REGION Network 77: WR 40001 - SETUP WRITING
   RUNG wire#powerrail
      { S7_Templates := "SrcType := Int" } EQ_Contact(in1 := "IEC_Counter_0_DB".CV, in2 := 71)
      Move(in := 16#8101, out1 => "Modbus_Send_Receive"."40001")
      { S7_Templates := "[card := 0, word_type := UInt, dword_type := UDInt, byte_type := USInt, any_type := Variant]" } "Modbus_Master_DB".Modbus_Master(REQ := wire#w1, MB_ADDR := 1, MODE := 1, DATA_ADDR := 40001, DATA_LEN := 1, DATA_PTR := "Modbus_Send_Receive"."40001", DONE => "Modbus".Done, BUSY => "Modbus".Busy, ERROR => "Modbus".Error, STATUS => "Modbus".Status)
   END_RUNG
   RUNG wire#powerrail
      Contact( "Comm_ok" )
      { S7_Templates := "SrcType := Int" } EQ_Contact(in1 := "IEC_Counter_0_DB".CV, in2 := 71)
      I_Contact( "Modbus_Master_DB".BUSY )
   END_RUNG wire#w1
   // the same network as SCL:
   IF "IEC_Counter_0_DB".CV = 71 THEN
       "Modbus_Send_Receive"."40001" := 16#8101;
       "Modbus_Master_DB"(REQ := "Comm_ok" AND ("IEC_Counter_0_DB".CV = 71) AND NOT "Modbus_Master_DB".BUSY,   // Modbus_Master
                          MB_ADDR := 1,
                          MODE := 1,
                          DATA_ADDR := 40001,
                          DATA_LEN := 1,
                          DATA_PTR := "Modbus_Send_Receive"."40001",
                          DONE => "Modbus".Done,
                          BUSY => "Modbus".Busy,
                          ERROR => "Modbus".Error,
                          STATUS => "Modbus".Status);
   END_IF;
END_REGION

REGION Network 78: WR 42001 - STS ON/OFF
   RUNG wire#powerrail
      { S7_Templates := "SrcType := Int" } EQ_Contact(in1 := "IEC_Counter_0_DB".CV, in2 := 72)
      { S7_Templates := "[card := 0, word_type := UInt, dword_type := UDInt, byte_type := USInt, any_type := Variant]" } "Modbus_Master_DB".Modbus_Master(REQ := wire#w2, MB_ADDR := 1, MODE := 1, DATA_ADDR := 42001, DATA_LEN := 1, DATA_PTR := "Modbus_Send_Receive"."42001", DONE => "Modbus".Done, BUSY => "Modbus".Busy, ERROR => "Modbus".Error, STATUS => "Modbus".Status)
   END_RUNG
   RUNG wire#powerrail
      Contact( "Liga_01" )
      Move(in := 16#0001, out1 => "Modbus_Send_Receive"."42001")
      wire#w1
      Contact( "Comm_ok" )
      { S7_Templates := "SrcType := Int" } EQ_Contact(in1 := "IEC_Counter_0_DB".CV, in2 := 72)
      I_Contact( "Modbus_Master_DB".BUSY )
   END_RUNG wire#w2
   RUNG wire#powerrail
      Contact( "Desliga_01" )
      Move(in := 16#0000, out1 => "Modbus_Send_Receive"."42001")
   END_RUNG wire#w1
   // the same network as SCL:
   IF "Liga_01" THEN "Modbus_Send_Receive"."42001" := 16#0001; END_IF;
   IF "Desliga_01" THEN "Modbus_Send_Receive"."42001" := 16#0000; END_IF;
   IF "IEC_Counter_0_DB".CV = 72 THEN
       "Modbus_Master_DB"(REQ := ("Liga_01" OR "Desliga_01") AND "Comm_ok" AND ("IEC_Counter_0_DB".CV = 72) AND NOT "Modbus_Master_DB".BUSY,   // Modbus_Master
                          MB_ADDR := 1,
                          MODE := 1,
                          DATA_ADDR := 42001,
                          DATA_LEN := 1,
                          DATA_PTR := "Modbus_Send_Receive"."42001",
                          DONE => "Modbus".Done,
                          BUSY => "Modbus".Busy,
                          ERROR => "Modbus".Error,
                          STATUS => "Modbus".Status);
   END_IF;
END_REGION

REGION Network 79: WR 42002 - OPER MODE
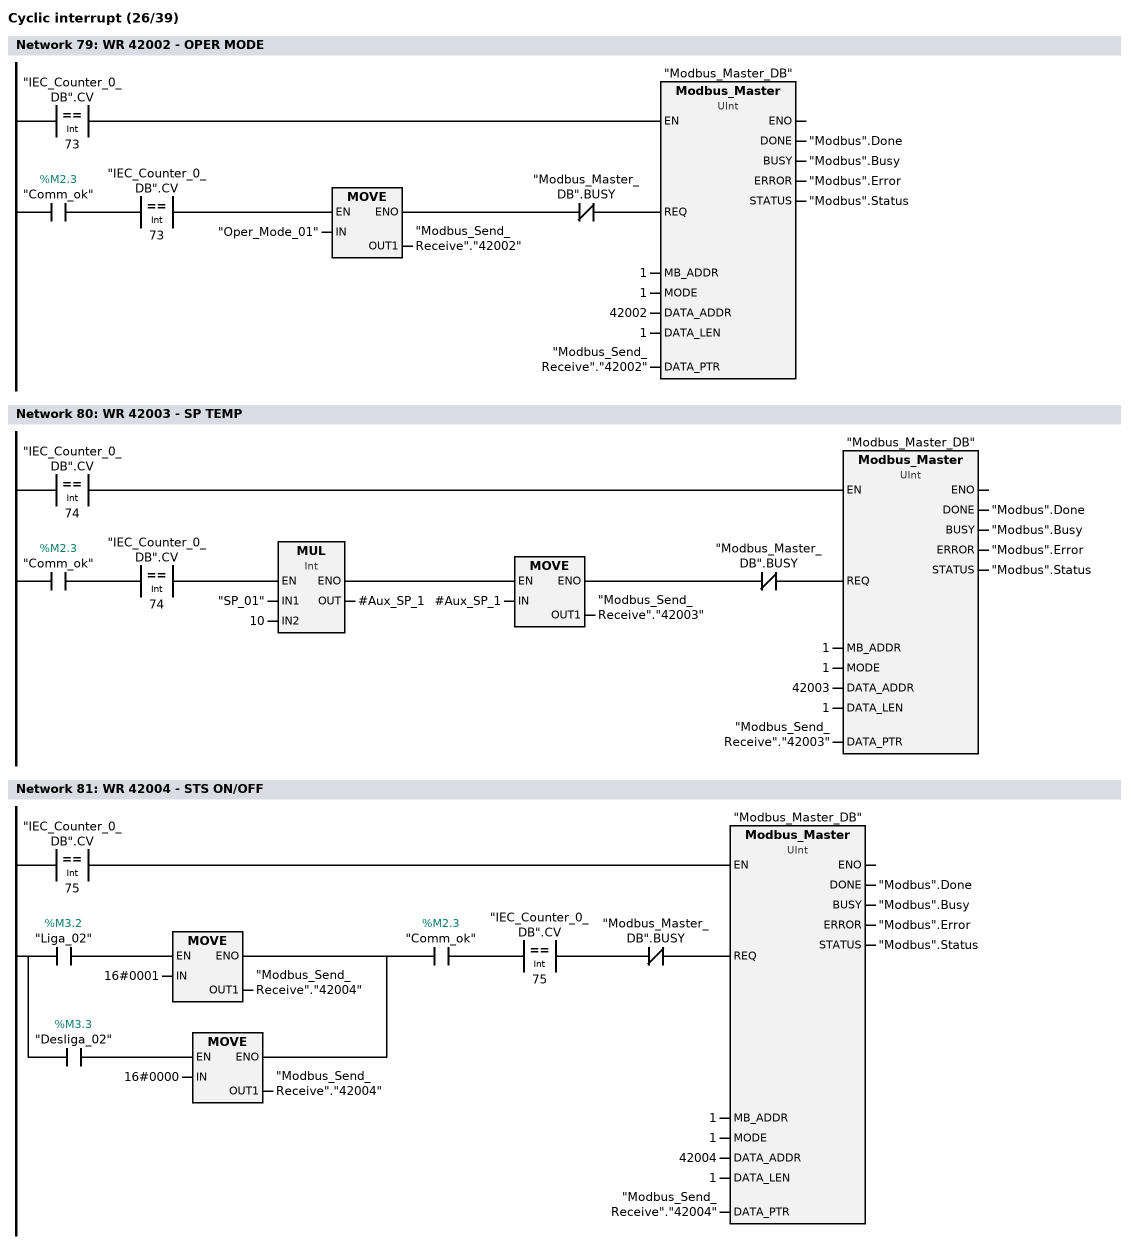
   RUNG wire#powerrail
      { S7_Templates := "SrcType := Int" } EQ_Contact(in1 := "IEC_Counter_0_DB".CV, in2 := 73)
      { S7_Templates := "[card := 0, word_type := UInt, dword_type := UDInt, byte_type := USInt, any_type := Variant]" } "Modbus_Master_DB".Modbus_Master(REQ := wire#w1, MB_ADDR := 1, MODE := 1, DATA_ADDR := 42002, DATA_LEN := 1, DATA_PTR := "Modbus_Send_Receive"."42002", DONE => "Modbus".Done, BUSY => "Modbus".Busy, ERROR => "Modbus".Error, STATUS => "Modbus".Status)
   END_RUNG
   RUNG wire#powerrail
      Contact( "Comm_ok" )
      { S7_Templates := "SrcType := Int" } EQ_Contact(in1 := "IEC_Counter_0_DB".CV, in2 := 73)
      Move(in := "Oper_Mode_01", out1 => "Modbus_Send_Receive"."42002")
      I_Contact( "Modbus_Master_DB".BUSY )
   END_RUNG wire#w1
   // the same network as SCL:
   #_w1 := "Comm_ok" AND ("IEC_Counter_0_DB".CV = 73);
   IF #_w1 THEN "Modbus_Send_Receive"."42002" := "Oper_Mode_01"; END_IF;
   IF "IEC_Counter_0_DB".CV = 73 THEN
       "Modbus_Master_DB"(REQ := #_w1 AND NOT "Modbus_Master_DB".BUSY,   // Modbus_Master
                          MB_ADDR := 1,
                          MODE := 1,
                          DATA_ADDR := 42002,
                          DATA_LEN := 1,
                          DATA_PTR := "Modbus_Send_Receive"."42002",
                          DONE => "Modbus".Done,
                          BUSY => "Modbus".Busy,
                          ERROR => "Modbus".Error,
                          STATUS => "Modbus".Status);
   END_IF;
END_REGION

REGION Network 80: WR 42003 - SP TEMP
   RUNG wire#powerrail
      { S7_Templates := "SrcType := Int" } EQ_Contact(in1 := "IEC_Counter_0_DB".CV, in2 := 74)
      { S7_Templates := "[card := 0, word_type := UInt, dword_type := UDInt, byte_type := USInt, any_type := Variant]" } "Modbus_Master_DB".Modbus_Master(REQ := wire#w1, MB_ADDR := 1, MODE := 1, DATA_ADDR := 42003, DATA_LEN := 1, DATA_PTR := "Modbus_Send_Receive"."42003", DONE => "Modbus".Done, BUSY => "Modbus".Busy, ERROR => "Modbus".Error, STATUS => "Modbus".Status)
   END_RUNG
   RUNG wire#powerrail
      Contact( "Comm_ok" )
      { S7_Templates := "SrcType := Int" } EQ_Contact(in1 := "IEC_Counter_0_DB".CV, in2 := 74)
      { S7_Templates := "SrcType := Int" } Mul(in1 := "SP_01", in2 := 10, out => #Aux_SP_1)
      Move(in := #Aux_SP_1, out1 => "Modbus_Send_Receive"."42003")
      I_Contact( "Modbus_Master_DB".BUSY )
   END_RUNG wire#w1
   // the same network as SCL:
   #_w1 := "Comm_ok" AND ("IEC_Counter_0_DB".CV = 74);
   IF #_w1 THEN
       #Aux_SP_1 := "SP_01" * 10;
       "Modbus_Send_Receive"."42003" := #Aux_SP_1;
   END_IF;
   IF "IEC_Counter_0_DB".CV = 74 THEN
       "Modbus_Master_DB"(REQ := #_w1 AND NOT "Modbus_Master_DB".BUSY,   // Modbus_Master
                          MB_ADDR := 1,
                          MODE := 1,
                          DATA_ADDR := 42003,
                          DATA_LEN := 1,
                          DATA_PTR := "Modbus_Send_Receive"."42003",
                          DONE => "Modbus".Done,
                          BUSY => "Modbus".Busy,
                          ERROR => "Modbus".Error,
                          STATUS => "Modbus".Status);
   END_IF;
END_REGION

REGION Network 81: WR 42004 - STS ON/OFF
   RUNG wire#powerrail
      { S7_Templates := "SrcType := Int" } EQ_Contact(in1 := "IEC_Counter_0_DB".CV, in2 := 75)
      { S7_Templates := "[card := 0, word_type := UInt, dword_type := UDInt, byte_type := USInt, any_type := Variant]" } "Modbus_Master_DB".Modbus_Master(REQ := wire#w2, MB_ADDR := 1, MODE := 1, DATA_ADDR := 42004, DATA_LEN := 1, DATA_PTR := "Modbus_Send_Receive"."42004", DONE => "Modbus".Done, BUSY => "Modbus".Busy, ERROR => "Modbus".Error, STATUS => "Modbus".Status)
   END_RUNG
   RUNG wire#powerrail
      Contact( "Liga_02" )
      Move(in := 16#0001, out1 => "Modbus_Send_Receive"."42004")
      wire#w1
      Contact( "Comm_ok" )
      { S7_Templates := "SrcType := Int" } EQ_Contact(in1 := "IEC_Counter_0_DB".CV, in2 := 75)
      I_Contact( "Modbus_Master_DB".BUSY )
   END_RUNG wire#w2
   RUNG wire#powerrail
      Contact( "Desliga_02" )
      Move(in := 16#0000, out1 => "Modbus_Send_Receive"."42004")
   END_RUNG wire#w1
   // the same network as SCL:
   IF "Liga_02" THEN "Modbus_Send_Receive"."42004" := 16#0001; END_IF;
   IF "Desliga_02" THEN "Modbus_Send_Receive"."42004" := 16#0000; END_IF;
   IF "IEC_Counter_0_DB".CV = 75 THEN
       "Modbus_Master_DB"(REQ := ("Liga_02" OR "Desliga_02") AND "Comm_ok" AND ("IEC_Counter_0_DB".CV = 75) AND NOT "Modbus_Master_DB".BUSY,   // Modbus_Master
                          MB_ADDR := 1,
                          MODE := 1,
                          DATA_ADDR := 42004,
                          DATA_LEN := 1,
                          DATA_PTR := "Modbus_Send_Receive"."42004",
                          DONE => "Modbus".Done,
                          BUSY => "Modbus".Busy,
                          ERROR => "Modbus".Error,
                          STATUS => "Modbus".Status);
   END_IF;
END_REGION

REGION Network 82: WR 42005 - OPER MODE
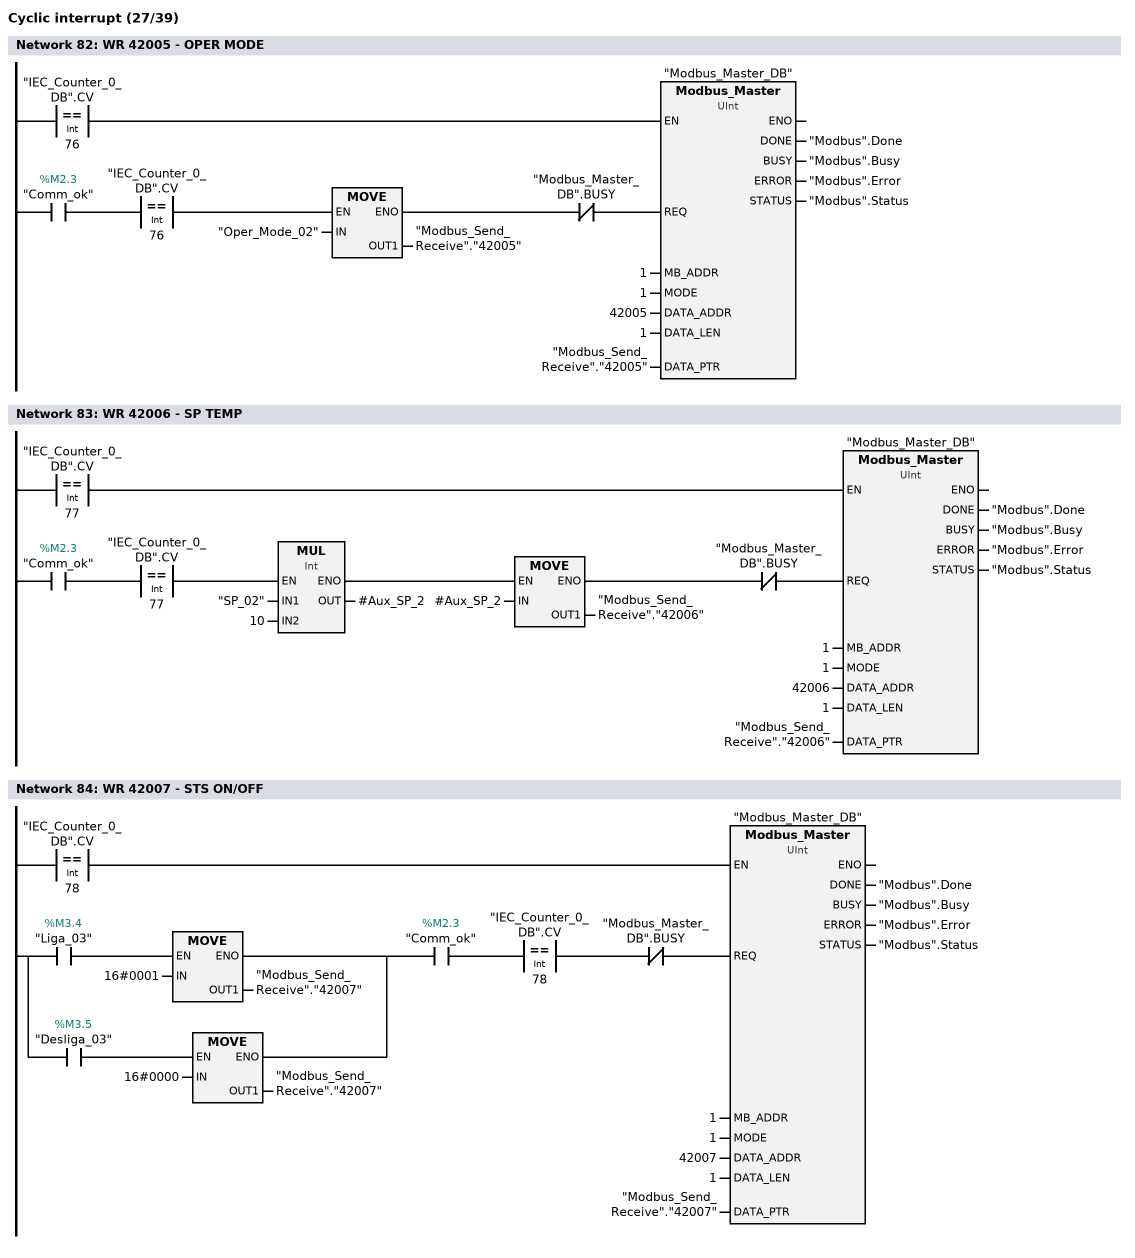
   RUNG wire#powerrail
      { S7_Templates := "SrcType := Int" } EQ_Contact(in1 := "IEC_Counter_0_DB".CV, in2 := 76)
      { S7_Templates := "[card := 0, word_type := UInt, dword_type := UDInt, byte_type := USInt, any_type := Variant]" } "Modbus_Master_DB".Modbus_Master(REQ := wire#w1, MB_ADDR := 1, MODE := 1, DATA_ADDR := 42005, DATA_LEN := 1, DATA_PTR := "Modbus_Send_Receive"."42005", DONE => "Modbus".Done, BUSY => "Modbus".Busy, ERROR => "Modbus".Error, STATUS => "Modbus".Status)
   END_RUNG
   RUNG wire#powerrail
      Contact( "Comm_ok" )
      { S7_Templates := "SrcType := Int" } EQ_Contact(in1 := "IEC_Counter_0_DB".CV, in2 := 76)
      Move(in := "Oper_Mode_02", out1 => "Modbus_Send_Receive"."42005")
      I_Contact( "Modbus_Master_DB".BUSY )
   END_RUNG wire#w1
   // the same network as SCL:
   #_w1 := "Comm_ok" AND ("IEC_Counter_0_DB".CV = 76);
   IF #_w1 THEN "Modbus_Send_Receive"."42005" := "Oper_Mode_02"; END_IF;
   IF "IEC_Counter_0_DB".CV = 76 THEN
       "Modbus_Master_DB"(REQ := #_w1 AND NOT "Modbus_Master_DB".BUSY,   // Modbus_Master
                          MB_ADDR := 1,
                          MODE := 1,
                          DATA_ADDR := 42005,
                          DATA_LEN := 1,
                          DATA_PTR := "Modbus_Send_Receive"."42005",
                          DONE => "Modbus".Done,
                          BUSY => "Modbus".Busy,
                          ERROR => "Modbus".Error,
                          STATUS => "Modbus".Status);
   END_IF;
END_REGION

REGION Network 83: WR 42006 - SP TEMP
   RUNG wire#powerrail
      { S7_Templates := "SrcType := Int" } EQ_Contact(in1 := "IEC_Counter_0_DB".CV, in2 := 77)
      { S7_Templates := "[card := 0, word_type := UInt, dword_type := UDInt, byte_type := USInt, any_type := Variant]" } "Modbus_Master_DB".Modbus_Master(REQ := wire#w1, MB_ADDR := 1, MODE := 1, DATA_ADDR := 42006, DATA_LEN := 1, DATA_PTR := "Modbus_Send_Receive"."42006", DONE => "Modbus".Done, BUSY => "Modbus".Busy, ERROR => "Modbus".Error, STATUS => "Modbus".Status)
   END_RUNG
   RUNG wire#powerrail
      Contact( "Comm_ok" )
      { S7_Templates := "SrcType := Int" } EQ_Contact(in1 := "IEC_Counter_0_DB".CV, in2 := 77)
      { S7_Templates := "SrcType := Int" } Mul(in1 := "SP_02", in2 := 10, out => #Aux_SP_2)
      Move(in := #Aux_SP_2, out1 => "Modbus_Send_Receive"."42006")
      I_Contact( "Modbus_Master_DB".BUSY )
   END_RUNG wire#w1
   // the same network as SCL:
   #_w1 := "Comm_ok" AND ("IEC_Counter_0_DB".CV = 77);
   IF #_w1 THEN
       #Aux_SP_2 := "SP_02" * 10;
       "Modbus_Send_Receive"."42006" := #Aux_SP_2;
   END_IF;
   IF "IEC_Counter_0_DB".CV = 77 THEN
       "Modbus_Master_DB"(REQ := #_w1 AND NOT "Modbus_Master_DB".BUSY,   // Modbus_Master
                          MB_ADDR := 1,
                          MODE := 1,
                          DATA_ADDR := 42006,
                          DATA_LEN := 1,
                          DATA_PTR := "Modbus_Send_Receive"."42006",
                          DONE => "Modbus".Done,
                          BUSY => "Modbus".Busy,
                          ERROR => "Modbus".Error,
                          STATUS => "Modbus".Status);
   END_IF;
END_REGION

REGION Network 84: WR 42007 - STS ON/OFF
   RUNG wire#powerrail
      { S7_Templates := "SrcType := Int" } EQ_Contact(in1 := "IEC_Counter_0_DB".CV, in2 := 78)
      { S7_Templates := "[card := 0, word_type := UInt, dword_type := UDInt, byte_type := USInt, any_type := Variant]" } "Modbus_Master_DB".Modbus_Master(REQ := wire#w2, MB_ADDR := 1, MODE := 1, DATA_ADDR := 42007, DATA_LEN := 1, DATA_PTR := "Modbus_Send_Receive"."42007", DONE => "Modbus".Done, BUSY => "Modbus".Busy, ERROR => "Modbus".Error, STATUS => "Modbus".Status)
   END_RUNG
   RUNG wire#powerrail
      Contact( "Liga_03" )
      Move(in := 16#0001, out1 => "Modbus_Send_Receive"."42007")
      wire#w1
      Contact( "Comm_ok" )
      { S7_Templates := "SrcType := Int" } EQ_Contact(in1 := "IEC_Counter_0_DB".CV, in2 := 78)
      I_Contact( "Modbus_Master_DB".BUSY )
   END_RUNG wire#w2
   RUNG wire#powerrail
      Contact( "Desliga_03" )
      Move(in := 16#0000, out1 => "Modbus_Send_Receive"."42007")
   END_RUNG wire#w1
   // the same network as SCL:
   IF "Liga_03" THEN "Modbus_Send_Receive"."42007" := 16#0001; END_IF;
   IF "Desliga_03" THEN "Modbus_Send_Receive"."42007" := 16#0000; END_IF;
   IF "IEC_Counter_0_DB".CV = 78 THEN
       "Modbus_Master_DB"(REQ := ("Liga_03" OR "Desliga_03") AND "Comm_ok" AND ("IEC_Counter_0_DB".CV = 78) AND NOT "Modbus_Master_DB".BUSY,   // Modbus_Master
                          MB_ADDR := 1,
                          MODE := 1,
                          DATA_ADDR := 42007,
                          DATA_LEN := 1,
                          DATA_PTR := "Modbus_Send_Receive"."42007",
                          DONE => "Modbus".Done,
                          BUSY => "Modbus".Busy,
                          ERROR => "Modbus".Error,
                          STATUS => "Modbus".Status);
   END_IF;
END_REGION

REGION Network 85: WR 42008 - OPER MODE
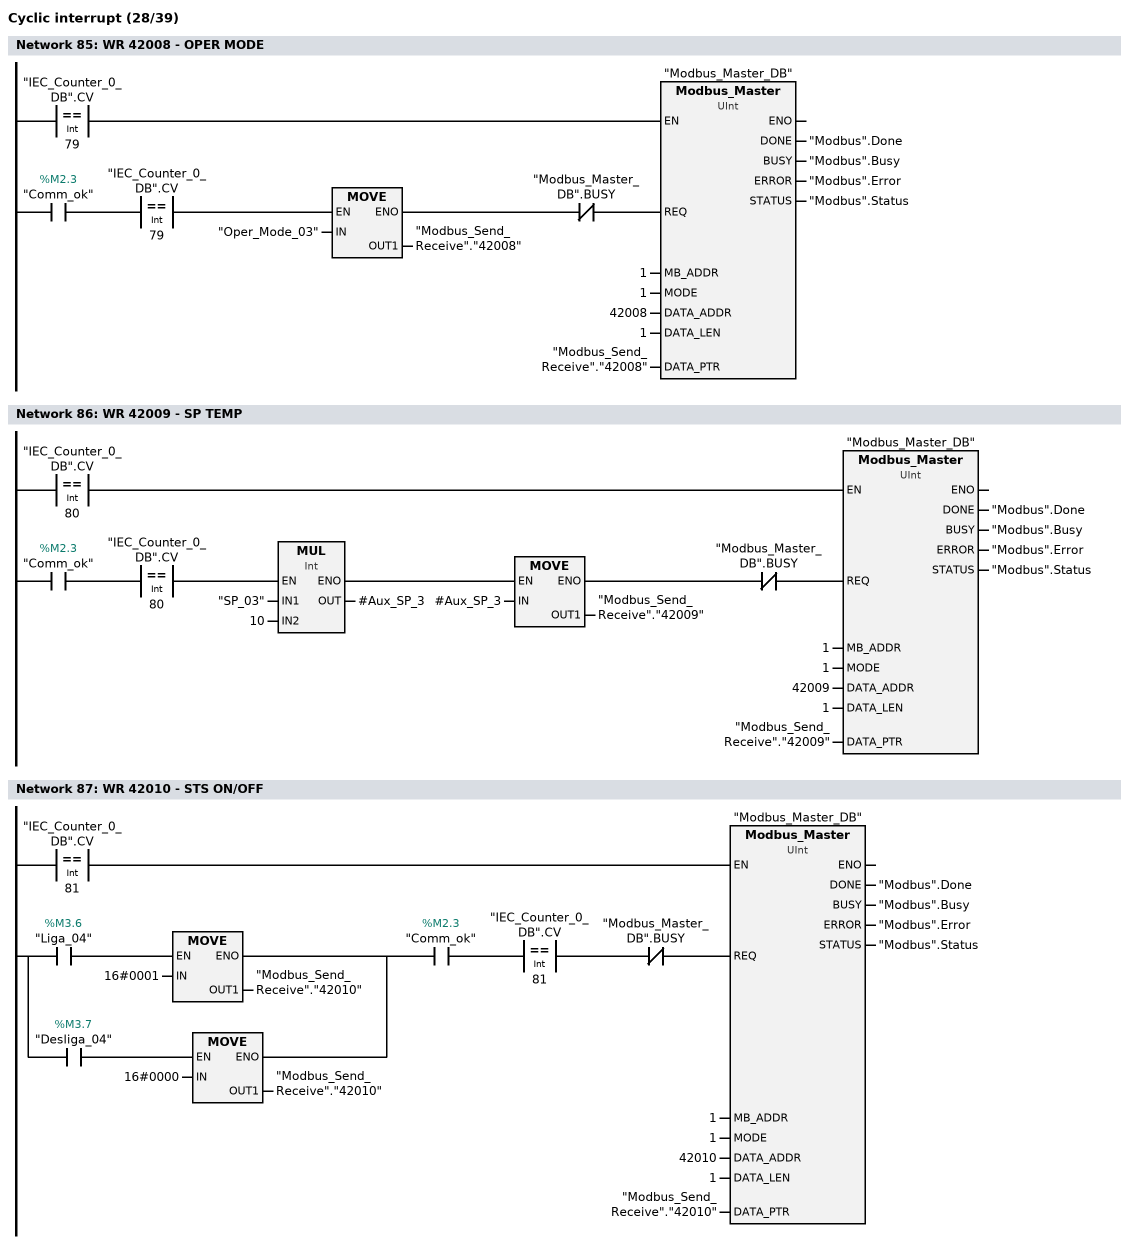
   RUNG wire#powerrail
      { S7_Templates := "SrcType := Int" } EQ_Contact(in1 := "IEC_Counter_0_DB".CV, in2 := 79)
      { S7_Templates := "[card := 0, word_type := UInt, dword_type := UDInt, byte_type := USInt, any_type := Variant]" } "Modbus_Master_DB".Modbus_Master(REQ := wire#w1, MB_ADDR := 1, MODE := 1, DATA_ADDR := 42008, DATA_LEN := 1, DATA_PTR := "Modbus_Send_Receive"."42008", DONE => "Modbus".Done, BUSY => "Modbus".Busy, ERROR => "Modbus".Error, STATUS => "Modbus".Status)
   END_RUNG
   RUNG wire#powerrail
      Contact( "Comm_ok" )
      { S7_Templates := "SrcType := Int" } EQ_Contact(in1 := "IEC_Counter_0_DB".CV, in2 := 79)
      Move(in := "Oper_Mode_03", out1 => "Modbus_Send_Receive"."42008")
      I_Contact( "Modbus_Master_DB".BUSY )
   END_RUNG wire#w1
   // the same network as SCL:
   #_w1 := "Comm_ok" AND ("IEC_Counter_0_DB".CV = 79);
   IF #_w1 THEN "Modbus_Send_Receive"."42008" := "Oper_Mode_03"; END_IF;
   IF "IEC_Counter_0_DB".CV = 79 THEN
       "Modbus_Master_DB"(REQ := #_w1 AND NOT "Modbus_Master_DB".BUSY,   // Modbus_Master
                          MB_ADDR := 1,
                          MODE := 1,
                          DATA_ADDR := 42008,
                          DATA_LEN := 1,
                          DATA_PTR := "Modbus_Send_Receive"."42008",
                          DONE => "Modbus".Done,
                          BUSY => "Modbus".Busy,
                          ERROR => "Modbus".Error,
                          STATUS => "Modbus".Status);
   END_IF;
END_REGION

REGION Network 86: WR 42009 - SP TEMP
   RUNG wire#powerrail
      { S7_Templates := "SrcType := Int" } EQ_Contact(in1 := "IEC_Counter_0_DB".CV, in2 := 80)
      { S7_Templates := "[card := 0, word_type := UInt, dword_type := UDInt, byte_type := USInt, any_type := Variant]" } "Modbus_Master_DB".Modbus_Master(REQ := wire#w1, MB_ADDR := 1, MODE := 1, DATA_ADDR := 42009, DATA_LEN := 1, DATA_PTR := "Modbus_Send_Receive"."42009", DONE => "Modbus".Done, BUSY => "Modbus".Busy, ERROR => "Modbus".Error, STATUS => "Modbus".Status)
   END_RUNG
   RUNG wire#powerrail
      Contact( "Comm_ok" )
      { S7_Templates := "SrcType := Int" } EQ_Contact(in1 := "IEC_Counter_0_DB".CV, in2 := 80)
      { S7_Templates := "SrcType := Int" } Mul(in1 := "SP_03", in2 := 10, out => #Aux_SP_3)
      Move(in := #Aux_SP_3, out1 => "Modbus_Send_Receive"."42009")
      I_Contact( "Modbus_Master_DB".BUSY )
   END_RUNG wire#w1
   // the same network as SCL:
   #_w1 := "Comm_ok" AND ("IEC_Counter_0_DB".CV = 80);
   IF #_w1 THEN
       #Aux_SP_3 := "SP_03" * 10;
       "Modbus_Send_Receive"."42009" := #Aux_SP_3;
   END_IF;
   IF "IEC_Counter_0_DB".CV = 80 THEN
       "Modbus_Master_DB"(REQ := #_w1 AND NOT "Modbus_Master_DB".BUSY,   // Modbus_Master
                          MB_ADDR := 1,
                          MODE := 1,
                          DATA_ADDR := 42009,
                          DATA_LEN := 1,
                          DATA_PTR := "Modbus_Send_Receive"."42009",
                          DONE => "Modbus".Done,
                          BUSY => "Modbus".Busy,
                          ERROR => "Modbus".Error,
                          STATUS => "Modbus".Status);
   END_IF;
END_REGION

REGION Network 87: WR 42010 - STS ON/OFF
   RUNG wire#powerrail
      { S7_Templates := "SrcType := Int" } EQ_Contact(in1 := "IEC_Counter_0_DB".CV, in2 := 81)
      { S7_Templates := "[card := 0, word_type := UInt, dword_type := UDInt, byte_type := USInt, any_type := Variant]" } "Modbus_Master_DB".Modbus_Master(REQ := wire#w2, MB_ADDR := 1, MODE := 1, DATA_ADDR := 42010, DATA_LEN := 1, DATA_PTR := "Modbus_Send_Receive"."42010", DONE => "Modbus".Done, BUSY => "Modbus".Busy, ERROR => "Modbus".Error, STATUS => "Modbus".Status)
   END_RUNG
   RUNG wire#powerrail
      Contact( "Liga_04" )
      Move(in := 16#0001, out1 => "Modbus_Send_Receive"."42010")
      wire#w1
      Contact( "Comm_ok" )
      { S7_Templates := "SrcType := Int" } EQ_Contact(in1 := "IEC_Counter_0_DB".CV, in2 := 81)
      I_Contact( "Modbus_Master_DB".BUSY )
   END_RUNG wire#w2
   RUNG wire#powerrail
      Contact( "Desliga_04" )
      Move(in := 16#0000, out1 => "Modbus_Send_Receive"."42010")
   END_RUNG wire#w1
   // the same network as SCL:
   IF "Liga_04" THEN "Modbus_Send_Receive"."42010" := 16#0001; END_IF;
   IF "Desliga_04" THEN "Modbus_Send_Receive"."42010" := 16#0000; END_IF;
   IF "IEC_Counter_0_DB".CV = 81 THEN
       "Modbus_Master_DB"(REQ := ("Liga_04" OR "Desliga_04") AND "Comm_ok" AND ("IEC_Counter_0_DB".CV = 81) AND NOT "Modbus_Master_DB".BUSY,   // Modbus_Master
                          MB_ADDR := 1,
                          MODE := 1,
                          DATA_ADDR := 42010,
                          DATA_LEN := 1,
                          DATA_PTR := "Modbus_Send_Receive"."42010",
                          DONE => "Modbus".Done,
                          BUSY => "Modbus".Busy,
                          ERROR => "Modbus".Error,
                          STATUS => "Modbus".Status);
   END_IF;
END_REGION

REGION Network 88: WR 42011 - OPER MODE
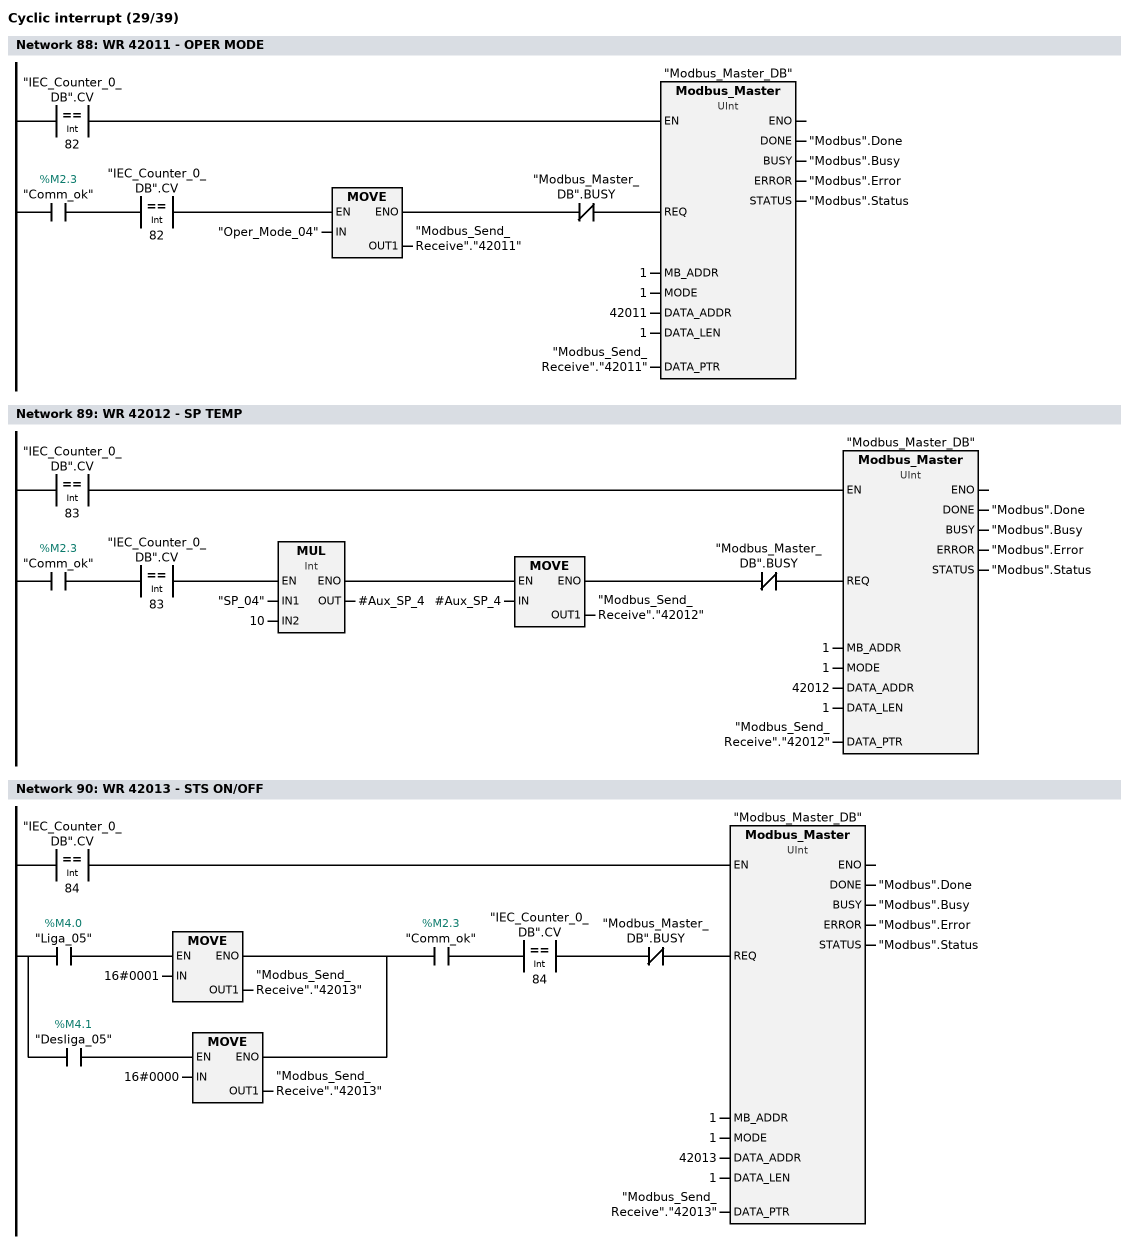
   RUNG wire#powerrail
      { S7_Templates := "SrcType := Int" } EQ_Contact(in1 := "IEC_Counter_0_DB".CV, in2 := 82)
      { S7_Templates := "[card := 0, word_type := UInt, dword_type := UDInt, byte_type := USInt, any_type := Variant]" } "Modbus_Master_DB".Modbus_Master(REQ := wire#w1, MB_ADDR := 1, MODE := 1, DATA_ADDR := 42011, DATA_LEN := 1, DATA_PTR := "Modbus_Send_Receive"."42011", DONE => "Modbus".Done, BUSY => "Modbus".Busy, ERROR => "Modbus".Error, STATUS => "Modbus".Status)
   END_RUNG
   RUNG wire#powerrail
      Contact( "Comm_ok" )
      { S7_Templates := "SrcType := Int" } EQ_Contact(in1 := "IEC_Counter_0_DB".CV, in2 := 82)
      Move(in := "Oper_Mode_04", out1 => "Modbus_Send_Receive"."42011")
      I_Contact( "Modbus_Master_DB".BUSY )
   END_RUNG wire#w1
   // the same network as SCL:
   #_w1 := "Comm_ok" AND ("IEC_Counter_0_DB".CV = 82);
   IF #_w1 THEN "Modbus_Send_Receive"."42011" := "Oper_Mode_04"; END_IF;
   IF "IEC_Counter_0_DB".CV = 82 THEN
       "Modbus_Master_DB"(REQ := #_w1 AND NOT "Modbus_Master_DB".BUSY,   // Modbus_Master
                          MB_ADDR := 1,
                          MODE := 1,
                          DATA_ADDR := 42011,
                          DATA_LEN := 1,
                          DATA_PTR := "Modbus_Send_Receive"."42011",
                          DONE => "Modbus".Done,
                          BUSY => "Modbus".Busy,
                          ERROR => "Modbus".Error,
                          STATUS => "Modbus".Status);
   END_IF;
END_REGION

REGION Network 89: WR 42012 - SP TEMP
   RUNG wire#powerrail
      { S7_Templates := "SrcType := Int" } EQ_Contact(in1 := "IEC_Counter_0_DB".CV, in2 := 83)
      { S7_Templates := "[card := 0, word_type := UInt, dword_type := UDInt, byte_type := USInt, any_type := Variant]" } "Modbus_Master_DB".Modbus_Master(REQ := wire#w1, MB_ADDR := 1, MODE := 1, DATA_ADDR := 42012, DATA_LEN := 1, DATA_PTR := "Modbus_Send_Receive"."42012", DONE => "Modbus".Done, BUSY => "Modbus".Busy, ERROR => "Modbus".Error, STATUS => "Modbus".Status)
   END_RUNG
   RUNG wire#powerrail
      Contact( "Comm_ok" )
      { S7_Templates := "SrcType := Int" } EQ_Contact(in1 := "IEC_Counter_0_DB".CV, in2 := 83)
      { S7_Templates := "SrcType := Int" } Mul(in1 := "SP_04", in2 := 10, out => #Aux_SP_4)
      Move(in := #Aux_SP_4, out1 => "Modbus_Send_Receive"."42012")
      I_Contact( "Modbus_Master_DB".BUSY )
   END_RUNG wire#w1
   // the same network as SCL:
   #_w1 := "Comm_ok" AND ("IEC_Counter_0_DB".CV = 83);
   IF #_w1 THEN
       #Aux_SP_4 := "SP_04" * 10;
       "Modbus_Send_Receive"."42012" := #Aux_SP_4;
   END_IF;
   IF "IEC_Counter_0_DB".CV = 83 THEN
       "Modbus_Master_DB"(REQ := #_w1 AND NOT "Modbus_Master_DB".BUSY,   // Modbus_Master
                          MB_ADDR := 1,
                          MODE := 1,
                          DATA_ADDR := 42012,
                          DATA_LEN := 1,
                          DATA_PTR := "Modbus_Send_Receive"."42012",
                          DONE => "Modbus".Done,
                          BUSY => "Modbus".Busy,
                          ERROR => "Modbus".Error,
                          STATUS => "Modbus".Status);
   END_IF;
END_REGION

REGION Network 90: WR 42013 - STS ON/OFF
   RUNG wire#powerrail
      { S7_Templates := "SrcType := Int" } EQ_Contact(in1 := "IEC_Counter_0_DB".CV, in2 := 84)
      { S7_Templates := "[card := 0, word_type := UInt, dword_type := UDInt, byte_type := USInt, any_type := Variant]" } "Modbus_Master_DB".Modbus_Master(REQ := wire#w2, MB_ADDR := 1, MODE := 1, DATA_ADDR := 42013, DATA_LEN := 1, DATA_PTR := "Modbus_Send_Receive"."42013", DONE => "Modbus".Done, BUSY => "Modbus".Busy, ERROR => "Modbus".Error, STATUS => "Modbus".Status)
   END_RUNG
   RUNG wire#powerrail
      Contact( "Liga_05" )
      Move(in := 16#0001, out1 => "Modbus_Send_Receive"."42013")
      wire#w1
      Contact( "Comm_ok" )
      { S7_Templates := "SrcType := Int" } EQ_Contact(in1 := "IEC_Counter_0_DB".CV, in2 := 84)
      I_Contact( "Modbus_Master_DB".BUSY )
   END_RUNG wire#w2
   RUNG wire#powerrail
      Contact( "Desliga_05" )
      Move(in := 16#0000, out1 => "Modbus_Send_Receive"."42013")
   END_RUNG wire#w1
   // the same network as SCL:
   IF "Liga_05" THEN "Modbus_Send_Receive"."42013" := 16#0001; END_IF;
   IF "Desliga_05" THEN "Modbus_Send_Receive"."42013" := 16#0000; END_IF;
   IF "IEC_Counter_0_DB".CV = 84 THEN
       "Modbus_Master_DB"(REQ := ("Liga_05" OR "Desliga_05") AND "Comm_ok" AND ("IEC_Counter_0_DB".CV = 84) AND NOT "Modbus_Master_DB".BUSY,   // Modbus_Master
                          MB_ADDR := 1,
                          MODE := 1,
                          DATA_ADDR := 42013,
                          DATA_LEN := 1,
                          DATA_PTR := "Modbus_Send_Receive"."42013",
                          DONE => "Modbus".Done,
                          BUSY => "Modbus".Busy,
                          ERROR => "Modbus".Error,
                          STATUS => "Modbus".Status);
   END_IF;
END_REGION

REGION Network 91: WR 42014 - OPER MODE
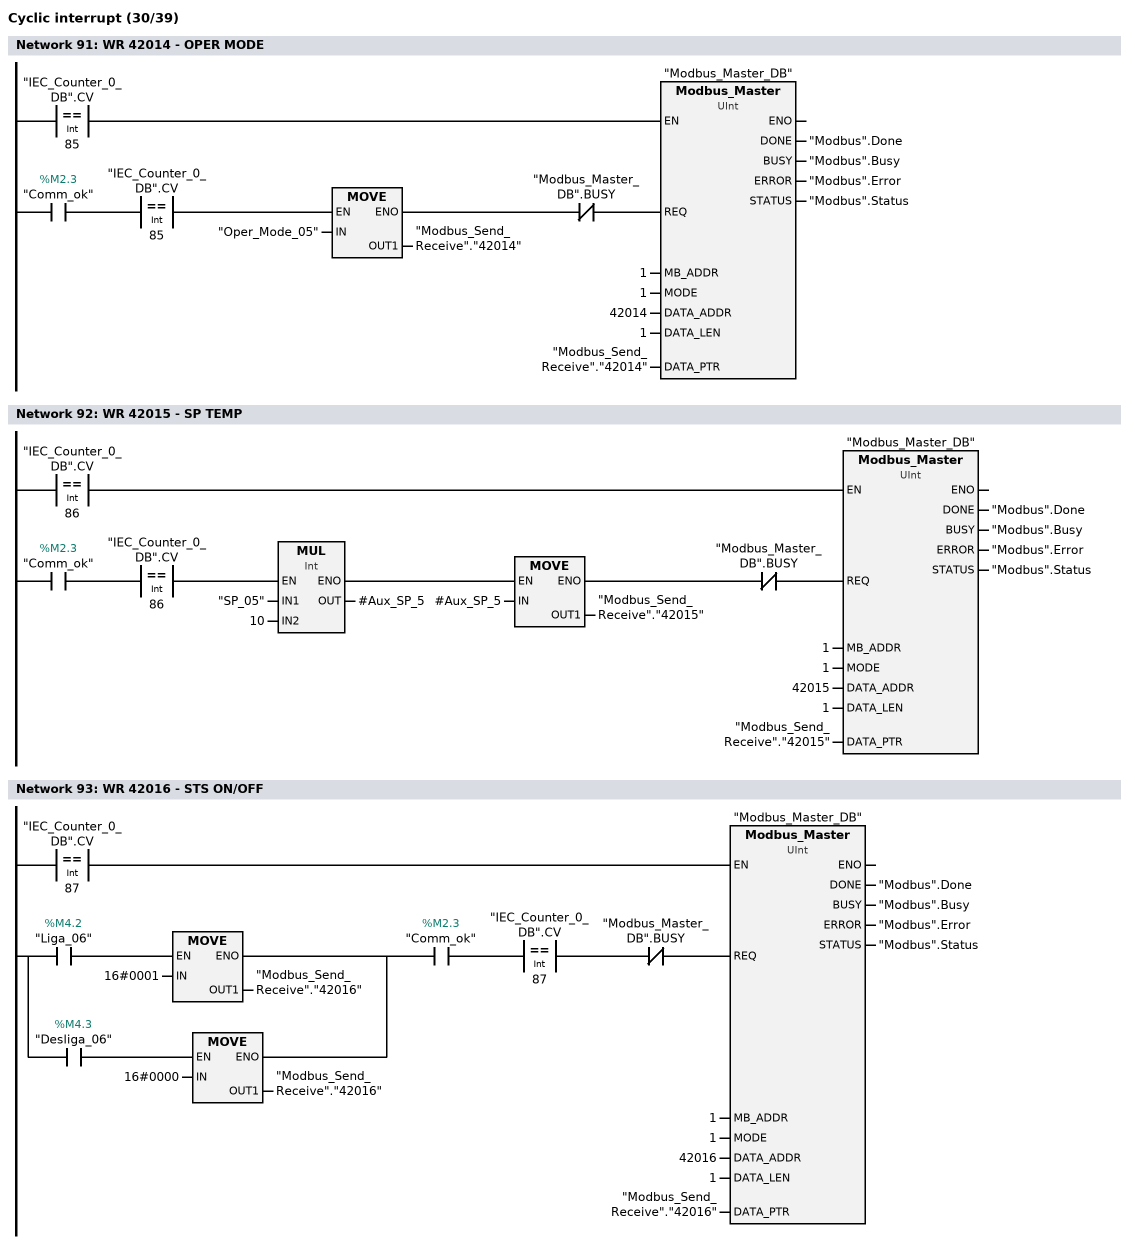
   RUNG wire#powerrail
      { S7_Templates := "SrcType := Int" } EQ_Contact(in1 := "IEC_Counter_0_DB".CV, in2 := 85)
      { S7_Templates := "[card := 0, word_type := UInt, dword_type := UDInt, byte_type := USInt, any_type := Variant]" } "Modbus_Master_DB".Modbus_Master(REQ := wire#w1, MB_ADDR := 1, MODE := 1, DATA_ADDR := 42014, DATA_LEN := 1, DATA_PTR := "Modbus_Send_Receive"."42014", DONE => "Modbus".Done, BUSY => "Modbus".Busy, ERROR => "Modbus".Error, STATUS => "Modbus".Status)
   END_RUNG
   RUNG wire#powerrail
      Contact( "Comm_ok" )
      { S7_Templates := "SrcType := Int" } EQ_Contact(in1 := "IEC_Counter_0_DB".CV, in2 := 85)
      Move(in := "Oper_Mode_05", out1 => "Modbus_Send_Receive"."42014")
      I_Contact( "Modbus_Master_DB".BUSY )
   END_RUNG wire#w1
   // the same network as SCL:
   #_w1 := "Comm_ok" AND ("IEC_Counter_0_DB".CV = 85);
   IF #_w1 THEN "Modbus_Send_Receive"."42014" := "Oper_Mode_05"; END_IF;
   IF "IEC_Counter_0_DB".CV = 85 THEN
       "Modbus_Master_DB"(REQ := #_w1 AND NOT "Modbus_Master_DB".BUSY,   // Modbus_Master
                          MB_ADDR := 1,
                          MODE := 1,
                          DATA_ADDR := 42014,
                          DATA_LEN := 1,
                          DATA_PTR := "Modbus_Send_Receive"."42014",
                          DONE => "Modbus".Done,
                          BUSY => "Modbus".Busy,
                          ERROR => "Modbus".Error,
                          STATUS => "Modbus".Status);
   END_IF;
END_REGION

REGION Network 92: WR 42015 - SP TEMP
   RUNG wire#powerrail
      { S7_Templates := "SrcType := Int" } EQ_Contact(in1 := "IEC_Counter_0_DB".CV, in2 := 86)
      { S7_Templates := "[card := 0, word_type := UInt, dword_type := UDInt, byte_type := USInt, any_type := Variant]" } "Modbus_Master_DB".Modbus_Master(REQ := wire#w1, MB_ADDR := 1, MODE := 1, DATA_ADDR := 42015, DATA_LEN := 1, DATA_PTR := "Modbus_Send_Receive"."42015", DONE => "Modbus".Done, BUSY => "Modbus".Busy, ERROR => "Modbus".Error, STATUS => "Modbus".Status)
   END_RUNG
   RUNG wire#powerrail
      Contact( "Comm_ok" )
      { S7_Templates := "SrcType := Int" } EQ_Contact(in1 := "IEC_Counter_0_DB".CV, in2 := 86)
      { S7_Templates := "SrcType := Int" } Mul(in1 := "SP_05", in2 := 10, out => #Aux_SP_5)
      Move(in := #Aux_SP_5, out1 => "Modbus_Send_Receive"."42015")
      I_Contact( "Modbus_Master_DB".BUSY )
   END_RUNG wire#w1
   // the same network as SCL:
   #_w1 := "Comm_ok" AND ("IEC_Counter_0_DB".CV = 86);
   IF #_w1 THEN
       #Aux_SP_5 := "SP_05" * 10;
       "Modbus_Send_Receive"."42015" := #Aux_SP_5;
   END_IF;
   IF "IEC_Counter_0_DB".CV = 86 THEN
       "Modbus_Master_DB"(REQ := #_w1 AND NOT "Modbus_Master_DB".BUSY,   // Modbus_Master
                          MB_ADDR := 1,
                          MODE := 1,
                          DATA_ADDR := 42015,
                          DATA_LEN := 1,
                          DATA_PTR := "Modbus_Send_Receive"."42015",
                          DONE => "Modbus".Done,
                          BUSY => "Modbus".Busy,
                          ERROR => "Modbus".Error,
                          STATUS => "Modbus".Status);
   END_IF;
END_REGION

REGION Network 93: WR 42016 - STS ON/OFF
   RUNG wire#powerrail
      { S7_Templates := "SrcType := Int" } EQ_Contact(in1 := "IEC_Counter_0_DB".CV, in2 := 87)
      { S7_Templates := "[card := 0, word_type := UInt, dword_type := UDInt, byte_type := USInt, any_type := Variant]" } "Modbus_Master_DB".Modbus_Master(REQ := wire#w2, MB_ADDR := 1, MODE := 1, DATA_ADDR := 42016, DATA_LEN := 1, DATA_PTR := "Modbus_Send_Receive"."42016", DONE => "Modbus".Done, BUSY => "Modbus".Busy, ERROR => "Modbus".Error, STATUS => "Modbus".Status)
   END_RUNG
   RUNG wire#powerrail
      Contact( "Liga_06" )
      Move(in := 16#0001, out1 => "Modbus_Send_Receive"."42016")
      wire#w1
      Contact( "Comm_ok" )
      { S7_Templates := "SrcType := Int" } EQ_Contact(in1 := "IEC_Counter_0_DB".CV, in2 := 87)
      I_Contact( "Modbus_Master_DB".BUSY )
   END_RUNG wire#w2
   RUNG wire#powerrail
      Contact( "Desliga_06" )
      Move(in := 16#0000, out1 => "Modbus_Send_Receive"."42016")
   END_RUNG wire#w1
   // the same network as SCL:
   IF "Liga_06" THEN "Modbus_Send_Receive"."42016" := 16#0001; END_IF;
   IF "Desliga_06" THEN "Modbus_Send_Receive"."42016" := 16#0000; END_IF;
   IF "IEC_Counter_0_DB".CV = 87 THEN
       "Modbus_Master_DB"(REQ := ("Liga_06" OR "Desliga_06") AND "Comm_ok" AND ("IEC_Counter_0_DB".CV = 87) AND NOT "Modbus_Master_DB".BUSY,   // Modbus_Master
                          MB_ADDR := 1,
                          MODE := 1,
                          DATA_ADDR := 42016,
                          DATA_LEN := 1,
                          DATA_PTR := "Modbus_Send_Receive"."42016",
                          DONE => "Modbus".Done,
                          BUSY => "Modbus".Busy,
                          ERROR => "Modbus".Error,
                          STATUS => "Modbus".Status);
   END_IF;
END_REGION

REGION Network 94: WR 42017 - OPER MODE
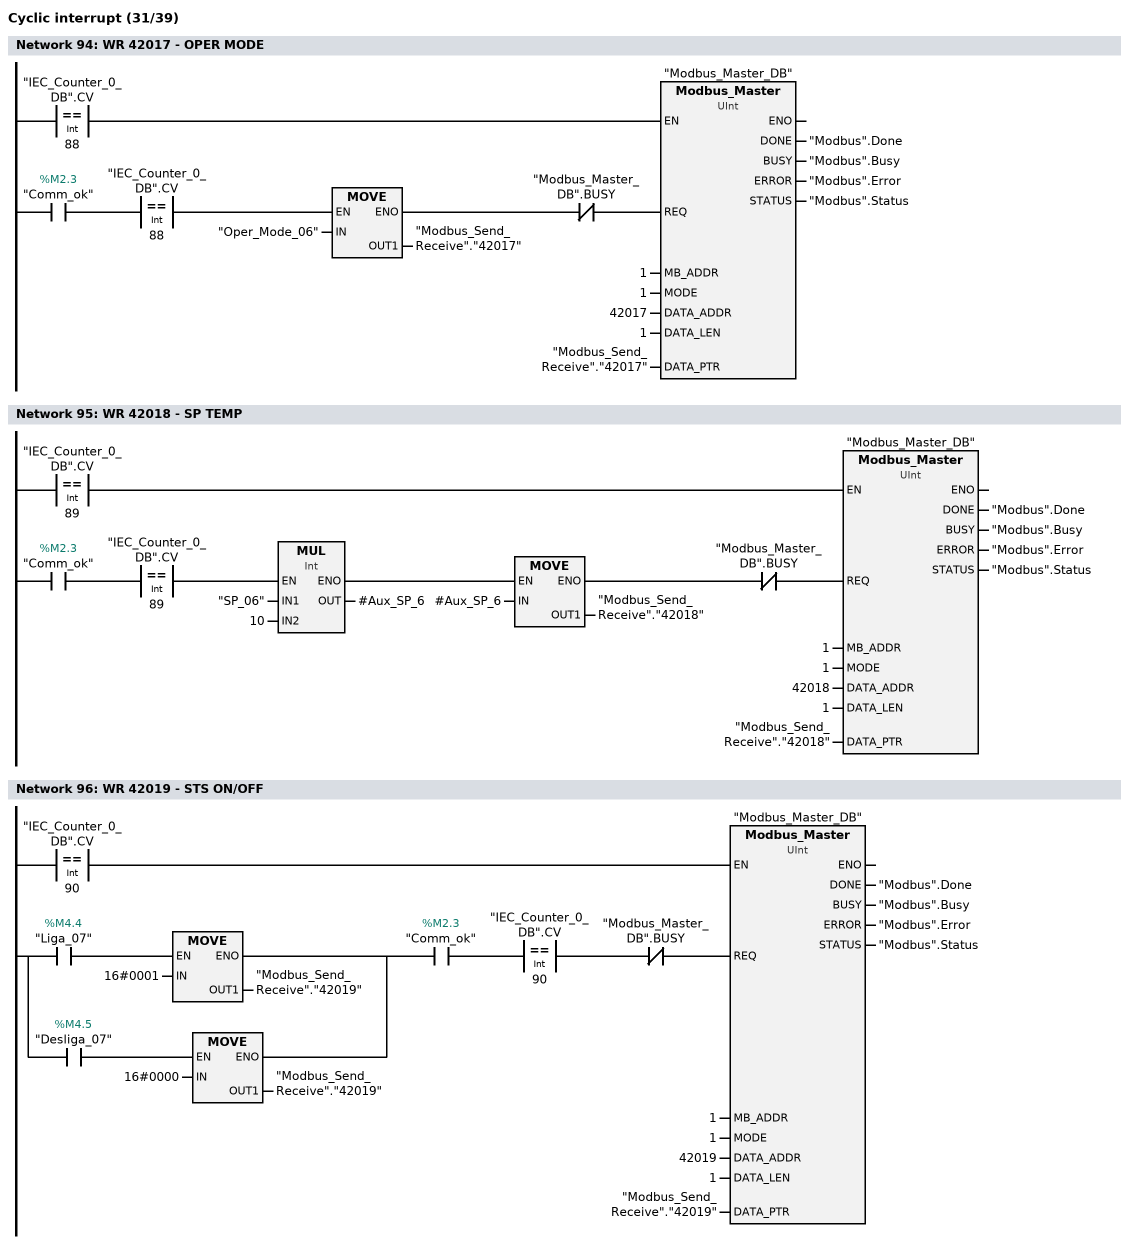
   RUNG wire#powerrail
      { S7_Templates := "SrcType := Int" } EQ_Contact(in1 := "IEC_Counter_0_DB".CV, in2 := 88)
      { S7_Templates := "[card := 0, word_type := UInt, dword_type := UDInt, byte_type := USInt, any_type := Variant]" } "Modbus_Master_DB".Modbus_Master(REQ := wire#w1, MB_ADDR := 1, MODE := 1, DATA_ADDR := 42017, DATA_LEN := 1, DATA_PTR := "Modbus_Send_Receive"."42017", DONE => "Modbus".Done, BUSY => "Modbus".Busy, ERROR => "Modbus".Error, STATUS => "Modbus".Status)
   END_RUNG
   RUNG wire#powerrail
      Contact( "Comm_ok" )
      { S7_Templates := "SrcType := Int" } EQ_Contact(in1 := "IEC_Counter_0_DB".CV, in2 := 88)
      Move(in := "Oper_Mode_06", out1 => "Modbus_Send_Receive"."42017")
      I_Contact( "Modbus_Master_DB".BUSY )
   END_RUNG wire#w1
   // the same network as SCL:
   #_w1 := "Comm_ok" AND ("IEC_Counter_0_DB".CV = 88);
   IF #_w1 THEN "Modbus_Send_Receive"."42017" := "Oper_Mode_06"; END_IF;
   IF "IEC_Counter_0_DB".CV = 88 THEN
       "Modbus_Master_DB"(REQ := #_w1 AND NOT "Modbus_Master_DB".BUSY,   // Modbus_Master
                          MB_ADDR := 1,
                          MODE := 1,
                          DATA_ADDR := 42017,
                          DATA_LEN := 1,
                          DATA_PTR := "Modbus_Send_Receive"."42017",
                          DONE => "Modbus".Done,
                          BUSY => "Modbus".Busy,
                          ERROR => "Modbus".Error,
                          STATUS => "Modbus".Status);
   END_IF;
END_REGION

REGION Network 95: WR 42018 - SP TEMP
   RUNG wire#powerrail
      { S7_Templates := "SrcType := Int" } EQ_Contact(in1 := "IEC_Counter_0_DB".CV, in2 := 89)
      { S7_Templates := "[card := 0, word_type := UInt, dword_type := UDInt, byte_type := USInt, any_type := Variant]" } "Modbus_Master_DB".Modbus_Master(REQ := wire#w1, MB_ADDR := 1, MODE := 1, DATA_ADDR := 42018, DATA_LEN := 1, DATA_PTR := "Modbus_Send_Receive"."42018", DONE => "Modbus".Done, BUSY => "Modbus".Busy, ERROR => "Modbus".Error, STATUS => "Modbus".Status)
   END_RUNG
   RUNG wire#powerrail
      Contact( "Comm_ok" )
      { S7_Templates := "SrcType := Int" } EQ_Contact(in1 := "IEC_Counter_0_DB".CV, in2 := 89)
      { S7_Templates := "SrcType := Int" } Mul(in1 := "SP_06", in2 := 10, out => #Aux_SP_6)
      Move(in := #Aux_SP_6, out1 => "Modbus_Send_Receive"."42018")
      I_Contact( "Modbus_Master_DB".BUSY )
   END_RUNG wire#w1
   // the same network as SCL:
   #_w1 := "Comm_ok" AND ("IEC_Counter_0_DB".CV = 89);
   IF #_w1 THEN
       #Aux_SP_6 := "SP_06" * 10;
       "Modbus_Send_Receive"."42018" := #Aux_SP_6;
   END_IF;
   IF "IEC_Counter_0_DB".CV = 89 THEN
       "Modbus_Master_DB"(REQ := #_w1 AND NOT "Modbus_Master_DB".BUSY,   // Modbus_Master
                          MB_ADDR := 1,
                          MODE := 1,
                          DATA_ADDR := 42018,
                          DATA_LEN := 1,
                          DATA_PTR := "Modbus_Send_Receive"."42018",
                          DONE => "Modbus".Done,
                          BUSY => "Modbus".Busy,
                          ERROR => "Modbus".Error,
                          STATUS => "Modbus".Status);
   END_IF;
END_REGION

REGION Network 96: WR 42019 - STS ON/OFF
   RUNG wire#powerrail
      { S7_Templates := "SrcType := Int" } EQ_Contact(in1 := "IEC_Counter_0_DB".CV, in2 := 90)
      { S7_Templates := "[card := 0, word_type := UInt, dword_type := UDInt, byte_type := USInt, any_type := Variant]" } "Modbus_Master_DB".Modbus_Master(REQ := wire#w2, MB_ADDR := 1, MODE := 1, DATA_ADDR := 42019, DATA_LEN := 1, DATA_PTR := "Modbus_Send_Receive"."42019", DONE => "Modbus".Done, BUSY => "Modbus".Busy, ERROR => "Modbus".Error, STATUS => "Modbus".Status)
   END_RUNG
   RUNG wire#powerrail
      Contact( "Liga_07" )
      Move(in := 16#0001, out1 => "Modbus_Send_Receive"."42019")
      wire#w1
      Contact( "Comm_ok" )
      { S7_Templates := "SrcType := Int" } EQ_Contact(in1 := "IEC_Counter_0_DB".CV, in2 := 90)
      I_Contact( "Modbus_Master_DB".BUSY )
   END_RUNG wire#w2
   RUNG wire#powerrail
      Contact( "Desliga_07" )
      Move(in := 16#0000, out1 => "Modbus_Send_Receive"."42019")
   END_RUNG wire#w1
   // the same network as SCL:
   IF "Liga_07" THEN "Modbus_Send_Receive"."42019" := 16#0001; END_IF;
   IF "Desliga_07" THEN "Modbus_Send_Receive"."42019" := 16#0000; END_IF;
   IF "IEC_Counter_0_DB".CV = 90 THEN
       "Modbus_Master_DB"(REQ := ("Liga_07" OR "Desliga_07") AND "Comm_ok" AND ("IEC_Counter_0_DB".CV = 90) AND NOT "Modbus_Master_DB".BUSY,   // Modbus_Master
                          MB_ADDR := 1,
                          MODE := 1,
                          DATA_ADDR := 42019,
                          DATA_LEN := 1,
                          DATA_PTR := "Modbus_Send_Receive"."42019",
                          DONE => "Modbus".Done,
                          BUSY => "Modbus".Busy,
                          ERROR => "Modbus".Error,
                          STATUS => "Modbus".Status);
   END_IF;
END_REGION

REGION Network 97: WR 42020 - OPER MODE
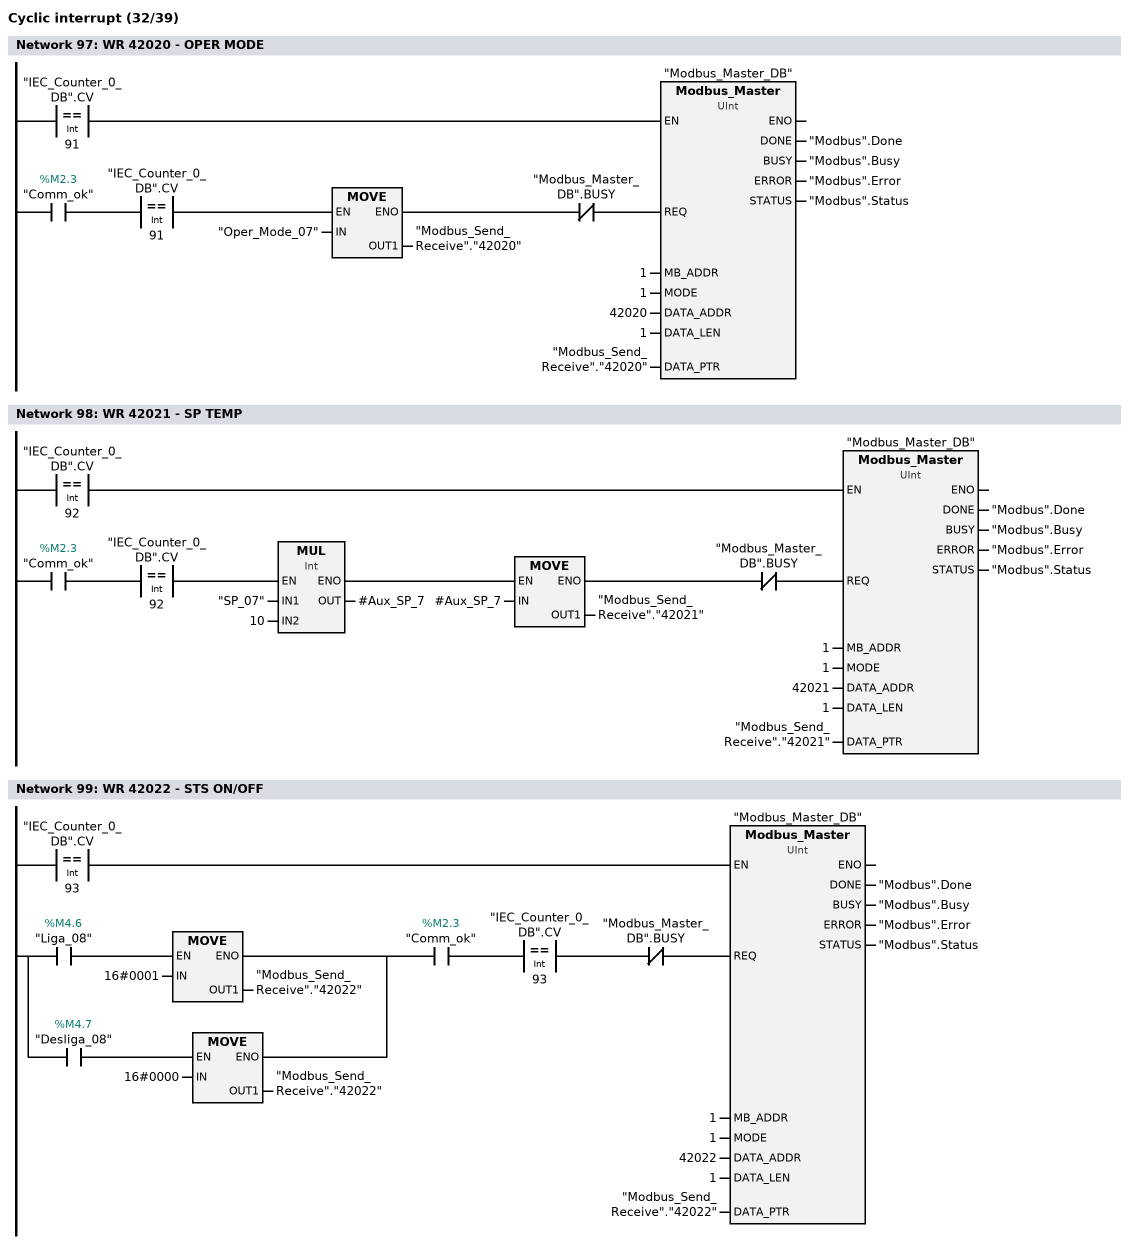
   RUNG wire#powerrail
      { S7_Templates := "SrcType := Int" } EQ_Contact(in1 := "IEC_Counter_0_DB".CV, in2 := 91)
      { S7_Templates := "[card := 0, word_type := UInt, dword_type := UDInt, byte_type := USInt, any_type := Variant]" } "Modbus_Master_DB".Modbus_Master(REQ := wire#w1, MB_ADDR := 1, MODE := 1, DATA_ADDR := 42020, DATA_LEN := 1, DATA_PTR := "Modbus_Send_Receive"."42020", DONE => "Modbus".Done, BUSY => "Modbus".Busy, ERROR => "Modbus".Error, STATUS => "Modbus".Status)
   END_RUNG
   RUNG wire#powerrail
      Contact( "Comm_ok" )
      { S7_Templates := "SrcType := Int" } EQ_Contact(in1 := "IEC_Counter_0_DB".CV, in2 := 91)
      Move(in := "Oper_Mode_07", out1 => "Modbus_Send_Receive"."42020")
      I_Contact( "Modbus_Master_DB".BUSY )
   END_RUNG wire#w1
   // the same network as SCL:
   #_w1 := "Comm_ok" AND ("IEC_Counter_0_DB".CV = 91);
   IF #_w1 THEN "Modbus_Send_Receive"."42020" := "Oper_Mode_07"; END_IF;
   IF "IEC_Counter_0_DB".CV = 91 THEN
       "Modbus_Master_DB"(REQ := #_w1 AND NOT "Modbus_Master_DB".BUSY,   // Modbus_Master
                          MB_ADDR := 1,
                          MODE := 1,
                          DATA_ADDR := 42020,
                          DATA_LEN := 1,
                          DATA_PTR := "Modbus_Send_Receive"."42020",
                          DONE => "Modbus".Done,
                          BUSY => "Modbus".Busy,
                          ERROR => "Modbus".Error,
                          STATUS => "Modbus".Status);
   END_IF;
END_REGION

REGION Network 98: WR 42021 - SP TEMP
   RUNG wire#powerrail
      { S7_Templates := "SrcType := Int" } EQ_Contact(in1 := "IEC_Counter_0_DB".CV, in2 := 92)
      { S7_Templates := "[card := 0, word_type := UInt, dword_type := UDInt, byte_type := USInt, any_type := Variant]" } "Modbus_Master_DB".Modbus_Master(REQ := wire#w1, MB_ADDR := 1, MODE := 1, DATA_ADDR := 42021, DATA_LEN := 1, DATA_PTR := "Modbus_Send_Receive"."42021", DONE => "Modbus".Done, BUSY => "Modbus".Busy, ERROR => "Modbus".Error, STATUS => "Modbus".Status)
   END_RUNG
   RUNG wire#powerrail
      Contact( "Comm_ok" )
      { S7_Templates := "SrcType := Int" } EQ_Contact(in1 := "IEC_Counter_0_DB".CV, in2 := 92)
      { S7_Templates := "SrcType := Int" } Mul(in1 := "SP_07", in2 := 10, out => #Aux_SP_7)
      Move(in := #Aux_SP_7, out1 => "Modbus_Send_Receive"."42021")
      I_Contact( "Modbus_Master_DB".BUSY )
   END_RUNG wire#w1
   // the same network as SCL:
   #_w1 := "Comm_ok" AND ("IEC_Counter_0_DB".CV = 92);
   IF #_w1 THEN
       #Aux_SP_7 := "SP_07" * 10;
       "Modbus_Send_Receive"."42021" := #Aux_SP_7;
   END_IF;
   IF "IEC_Counter_0_DB".CV = 92 THEN
       "Modbus_Master_DB"(REQ := #_w1 AND NOT "Modbus_Master_DB".BUSY,   // Modbus_Master
                          MB_ADDR := 1,
                          MODE := 1,
                          DATA_ADDR := 42021,
                          DATA_LEN := 1,
                          DATA_PTR := "Modbus_Send_Receive"."42021",
                          DONE => "Modbus".Done,
                          BUSY => "Modbus".Busy,
                          ERROR => "Modbus".Error,
                          STATUS => "Modbus".Status);
   END_IF;
END_REGION

REGION Network 99: WR 42022 - STS ON/OFF
   RUNG wire#powerrail
      { S7_Templates := "SrcType := Int" } EQ_Contact(in1 := "IEC_Counter_0_DB".CV, in2 := 93)
      { S7_Templates := "[card := 0, word_type := UInt, dword_type := UDInt, byte_type := USInt, any_type := Variant]" } "Modbus_Master_DB".Modbus_Master(REQ := wire#w2, MB_ADDR := 1, MODE := 1, DATA_ADDR := 42022, DATA_LEN := 1, DATA_PTR := "Modbus_Send_Receive"."42022", DONE => "Modbus".Done, BUSY => "Modbus".Busy, ERROR => "Modbus".Error, STATUS => "Modbus".Status)
   END_RUNG
   RUNG wire#powerrail
      Contact( "Liga_08" )
      Move(in := 16#0001, out1 => "Modbus_Send_Receive"."42022")
      wire#w1
      Contact( "Comm_ok" )
      { S7_Templates := "SrcType := Int" } EQ_Contact(in1 := "IEC_Counter_0_DB".CV, in2 := 93)
      I_Contact( "Modbus_Master_DB".BUSY )
   END_RUNG wire#w2
   RUNG wire#powerrail
      Contact( "Desliga_08" )
      Move(in := 16#0000, out1 => "Modbus_Send_Receive"."42022")
   END_RUNG wire#w1
   // the same network as SCL:
   IF "Liga_08" THEN "Modbus_Send_Receive"."42022" := 16#0001; END_IF;
   IF "Desliga_08" THEN "Modbus_Send_Receive"."42022" := 16#0000; END_IF;
   IF "IEC_Counter_0_DB".CV = 93 THEN
       "Modbus_Master_DB"(REQ := ("Liga_08" OR "Desliga_08") AND "Comm_ok" AND ("IEC_Counter_0_DB".CV = 93) AND NOT "Modbus_Master_DB".BUSY,   // Modbus_Master
                          MB_ADDR := 1,
                          MODE := 1,
                          DATA_ADDR := 42022,
                          DATA_LEN := 1,
                          DATA_PTR := "Modbus_Send_Receive"."42022",
                          DONE => "Modbus".Done,
                          BUSY => "Modbus".Busy,
                          ERROR => "Modbus".Error,
                          STATUS => "Modbus".Status);
   END_IF;
END_REGION

REGION Network 100: WR 42023 - OPER MODE
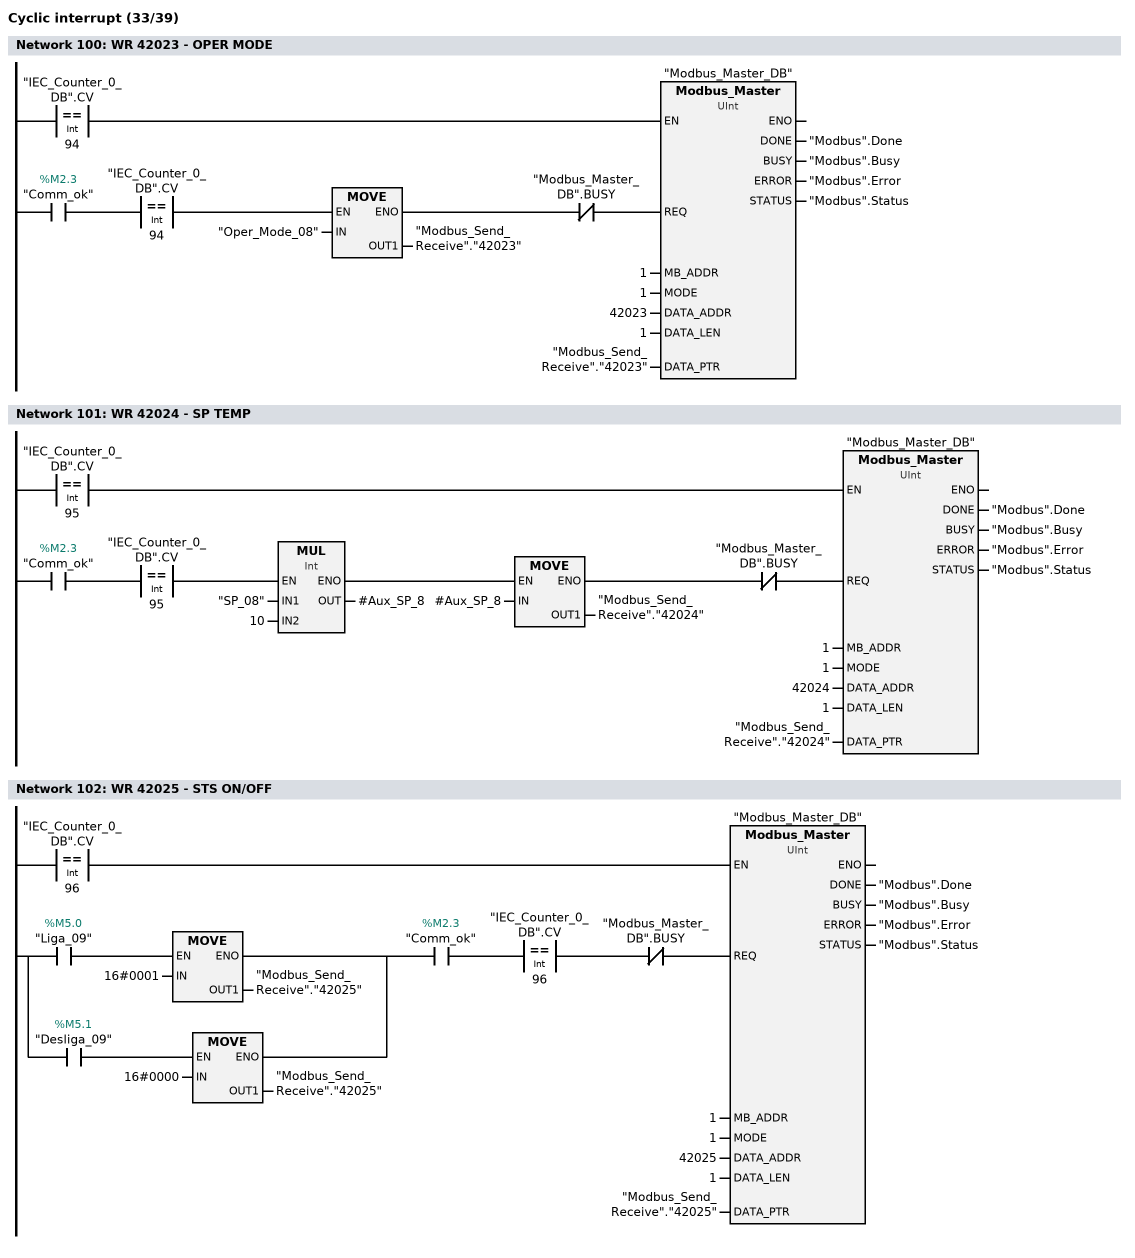
   RUNG wire#powerrail
      { S7_Templates := "SrcType := Int" } EQ_Contact(in1 := "IEC_Counter_0_DB".CV, in2 := 94)
      { S7_Templates := "[card := 0, word_type := UInt, dword_type := UDInt, byte_type := USInt, any_type := Variant]" } "Modbus_Master_DB".Modbus_Master(REQ := wire#w1, MB_ADDR := 1, MODE := 1, DATA_ADDR := 42023, DATA_LEN := 1, DATA_PTR := "Modbus_Send_Receive"."42023", DONE => "Modbus".Done, BUSY => "Modbus".Busy, ERROR => "Modbus".Error, STATUS => "Modbus".Status)
   END_RUNG
   RUNG wire#powerrail
      Contact( "Comm_ok" )
      { S7_Templates := "SrcType := Int" } EQ_Contact(in1 := "IEC_Counter_0_DB".CV, in2 := 94)
      Move(in := "Oper_Mode_08", out1 => "Modbus_Send_Receive"."42023")
      I_Contact( "Modbus_Master_DB".BUSY )
   END_RUNG wire#w1
   // the same network as SCL:
   #_w1 := "Comm_ok" AND ("IEC_Counter_0_DB".CV = 94);
   IF #_w1 THEN "Modbus_Send_Receive"."42023" := "Oper_Mode_08"; END_IF;
   IF "IEC_Counter_0_DB".CV = 94 THEN
       "Modbus_Master_DB"(REQ := #_w1 AND NOT "Modbus_Master_DB".BUSY,   // Modbus_Master
                          MB_ADDR := 1,
                          MODE := 1,
                          DATA_ADDR := 42023,
                          DATA_LEN := 1,
                          DATA_PTR := "Modbus_Send_Receive"."42023",
                          DONE => "Modbus".Done,
                          BUSY => "Modbus".Busy,
                          ERROR => "Modbus".Error,
                          STATUS => "Modbus".Status);
   END_IF;
END_REGION

REGION Network 101: WR 42024 - SP TEMP
   RUNG wire#powerrail
      { S7_Templates := "SrcType := Int" } EQ_Contact(in1 := "IEC_Counter_0_DB".CV, in2 := 95)
      { S7_Templates := "[card := 0, word_type := UInt, dword_type := UDInt, byte_type := USInt, any_type := Variant]" } "Modbus_Master_DB".Modbus_Master(REQ := wire#w1, MB_ADDR := 1, MODE := 1, DATA_ADDR := 42024, DATA_LEN := 1, DATA_PTR := "Modbus_Send_Receive"."42024", DONE => "Modbus".Done, BUSY => "Modbus".Busy, ERROR => "Modbus".Error, STATUS => "Modbus".Status)
   END_RUNG
   RUNG wire#powerrail
      Contact( "Comm_ok" )
      { S7_Templates := "SrcType := Int" } EQ_Contact(in1 := "IEC_Counter_0_DB".CV, in2 := 95)
      { S7_Templates := "SrcType := Int" } Mul(in1 := "SP_08", in2 := 10, out => #Aux_SP_8)
      Move(in := #Aux_SP_8, out1 => "Modbus_Send_Receive"."42024")
      I_Contact( "Modbus_Master_DB".BUSY )
   END_RUNG wire#w1
   // the same network as SCL:
   #_w1 := "Comm_ok" AND ("IEC_Counter_0_DB".CV = 95);
   IF #_w1 THEN
       #Aux_SP_8 := "SP_08" * 10;
       "Modbus_Send_Receive"."42024" := #Aux_SP_8;
   END_IF;
   IF "IEC_Counter_0_DB".CV = 95 THEN
       "Modbus_Master_DB"(REQ := #_w1 AND NOT "Modbus_Master_DB".BUSY,   // Modbus_Master
                          MB_ADDR := 1,
                          MODE := 1,
                          DATA_ADDR := 42024,
                          DATA_LEN := 1,
                          DATA_PTR := "Modbus_Send_Receive"."42024",
                          DONE => "Modbus".Done,
                          BUSY => "Modbus".Busy,
                          ERROR => "Modbus".Error,
                          STATUS => "Modbus".Status);
   END_IF;
END_REGION

REGION Network 102: WR 42025 - STS ON/OFF
   RUNG wire#powerrail
      { S7_Templates := "SrcType := Int" } EQ_Contact(in1 := "IEC_Counter_0_DB".CV, in2 := 96)
      { S7_Templates := "[card := 0, word_type := UInt, dword_type := UDInt, byte_type := USInt, any_type := Variant]" } "Modbus_Master_DB".Modbus_Master(REQ := wire#w2, MB_ADDR := 1, MODE := 1, DATA_ADDR := 42025, DATA_LEN := 1, DATA_PTR := "Modbus_Send_Receive"."42025", DONE => "Modbus".Done, BUSY => "Modbus".Busy, ERROR => "Modbus".Error, STATUS => "Modbus".Status)
   END_RUNG
   RUNG wire#powerrail
      Contact( "Liga_09" )
      Move(in := 16#0001, out1 => "Modbus_Send_Receive"."42025")
      wire#w1
      Contact( "Comm_ok" )
      { S7_Templates := "SrcType := Int" } EQ_Contact(in1 := "IEC_Counter_0_DB".CV, in2 := 96)
      I_Contact( "Modbus_Master_DB".BUSY )
   END_RUNG wire#w2
   RUNG wire#powerrail
      Contact( "Desliga_09" )
      Move(in := 16#0000, out1 => "Modbus_Send_Receive"."42025")
   END_RUNG wire#w1
   // the same network as SCL:
   IF "Liga_09" THEN "Modbus_Send_Receive"."42025" := 16#0001; END_IF;
   IF "Desliga_09" THEN "Modbus_Send_Receive"."42025" := 16#0000; END_IF;
   IF "IEC_Counter_0_DB".CV = 96 THEN
       "Modbus_Master_DB"(REQ := ("Liga_09" OR "Desliga_09") AND "Comm_ok" AND ("IEC_Counter_0_DB".CV = 96) AND NOT "Modbus_Master_DB".BUSY,   // Modbus_Master
                          MB_ADDR := 1,
                          MODE := 1,
                          DATA_ADDR := 42025,
                          DATA_LEN := 1,
                          DATA_PTR := "Modbus_Send_Receive"."42025",
                          DONE => "Modbus".Done,
                          BUSY => "Modbus".Busy,
                          ERROR => "Modbus".Error,
                          STATUS => "Modbus".Status);
   END_IF;
END_REGION

REGION Network 103: WR 42026 - OPER MODE
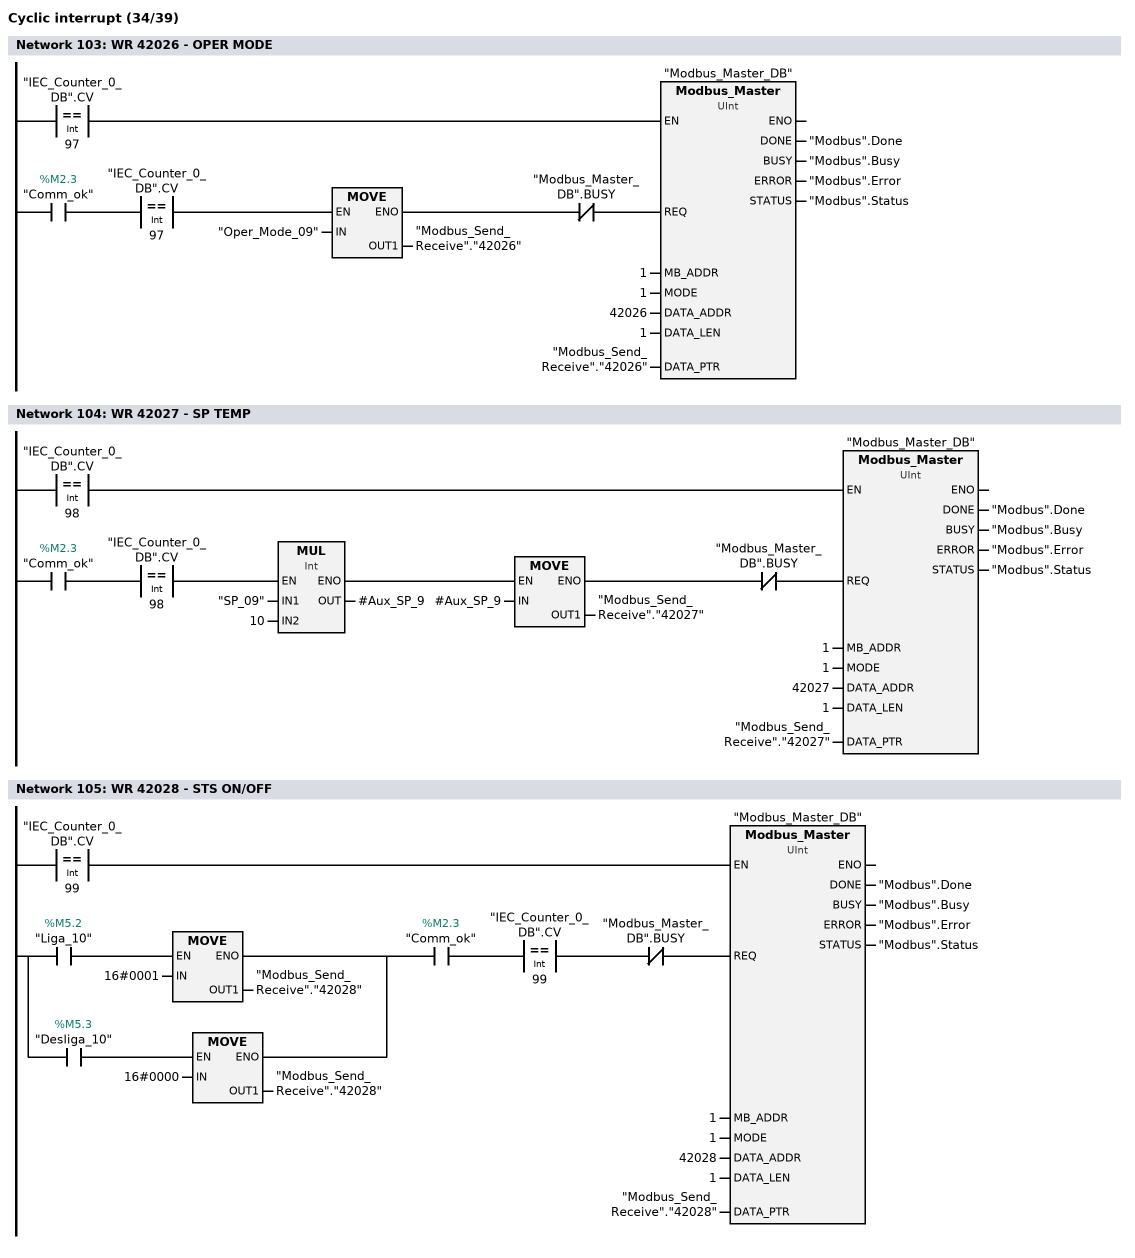
   RUNG wire#powerrail
      { S7_Templates := "SrcType := Int" } EQ_Contact(in1 := "IEC_Counter_0_DB".CV, in2 := 97)
      { S7_Templates := "[card := 0, word_type := UInt, dword_type := UDInt, byte_type := USInt, any_type := Variant]" } "Modbus_Master_DB".Modbus_Master(REQ := wire#w1, MB_ADDR := 1, MODE := 1, DATA_ADDR := 42026, DATA_LEN := 1, DATA_PTR := "Modbus_Send_Receive"."42026", DONE => "Modbus".Done, BUSY => "Modbus".Busy, ERROR => "Modbus".Error, STATUS => "Modbus".Status)
   END_RUNG
   RUNG wire#powerrail
      Contact( "Comm_ok" )
      { S7_Templates := "SrcType := Int" } EQ_Contact(in1 := "IEC_Counter_0_DB".CV, in2 := 97)
      Move(in := "Oper_Mode_09", out1 => "Modbus_Send_Receive"."42026")
      I_Contact( "Modbus_Master_DB".BUSY )
   END_RUNG wire#w1
   // the same network as SCL:
   #_w1 := "Comm_ok" AND ("IEC_Counter_0_DB".CV = 97);
   IF #_w1 THEN "Modbus_Send_Receive"."42026" := "Oper_Mode_09"; END_IF;
   IF "IEC_Counter_0_DB".CV = 97 THEN
       "Modbus_Master_DB"(REQ := #_w1 AND NOT "Modbus_Master_DB".BUSY,   // Modbus_Master
                          MB_ADDR := 1,
                          MODE := 1,
                          DATA_ADDR := 42026,
                          DATA_LEN := 1,
                          DATA_PTR := "Modbus_Send_Receive"."42026",
                          DONE => "Modbus".Done,
                          BUSY => "Modbus".Busy,
                          ERROR => "Modbus".Error,
                          STATUS => "Modbus".Status);
   END_IF;
END_REGION

REGION Network 104: WR 42027 - SP TEMP
   RUNG wire#powerrail
      { S7_Templates := "SrcType := Int" } EQ_Contact(in1 := "IEC_Counter_0_DB".CV, in2 := 98)
      { S7_Templates := "[card := 0, word_type := UInt, dword_type := UDInt, byte_type := USInt, any_type := Variant]" } "Modbus_Master_DB".Modbus_Master(REQ := wire#w1, MB_ADDR := 1, MODE := 1, DATA_ADDR := 42027, DATA_LEN := 1, DATA_PTR := "Modbus_Send_Receive"."42027", DONE => "Modbus".Done, BUSY => "Modbus".Busy, ERROR => "Modbus".Error, STATUS => "Modbus".Status)
   END_RUNG
   RUNG wire#powerrail
      Contact( "Comm_ok" )
      { S7_Templates := "SrcType := Int" } EQ_Contact(in1 := "IEC_Counter_0_DB".CV, in2 := 98)
      { S7_Templates := "SrcType := Int" } Mul(in1 := "SP_09", in2 := 10, out => #Aux_SP_9)
      Move(in := #Aux_SP_9, out1 => "Modbus_Send_Receive"."42027")
      I_Contact( "Modbus_Master_DB".BUSY )
   END_RUNG wire#w1
   // the same network as SCL:
   #_w1 := "Comm_ok" AND ("IEC_Counter_0_DB".CV = 98);
   IF #_w1 THEN
       #Aux_SP_9 := "SP_09" * 10;
       "Modbus_Send_Receive"."42027" := #Aux_SP_9;
   END_IF;
   IF "IEC_Counter_0_DB".CV = 98 THEN
       "Modbus_Master_DB"(REQ := #_w1 AND NOT "Modbus_Master_DB".BUSY,   // Modbus_Master
                          MB_ADDR := 1,
                          MODE := 1,
                          DATA_ADDR := 42027,
                          DATA_LEN := 1,
                          DATA_PTR := "Modbus_Send_Receive"."42027",
                          DONE => "Modbus".Done,
                          BUSY => "Modbus".Busy,
                          ERROR => "Modbus".Error,
                          STATUS => "Modbus".Status);
   END_IF;
END_REGION

REGION Network 105: WR 42028 - STS ON/OFF
   RUNG wire#powerrail
      { S7_Templates := "SrcType := Int" } EQ_Contact(in1 := "IEC_Counter_0_DB".CV, in2 := 99)
      { S7_Templates := "[card := 0, word_type := UInt, dword_type := UDInt, byte_type := USInt, any_type := Variant]" } "Modbus_Master_DB".Modbus_Master(REQ := wire#w2, MB_ADDR := 1, MODE := 1, DATA_ADDR := 42028, DATA_LEN := 1, DATA_PTR := "Modbus_Send_Receive"."42028", DONE => "Modbus".Done, BUSY => "Modbus".Busy, ERROR => "Modbus".Error, STATUS => "Modbus".Status)
   END_RUNG
   RUNG wire#powerrail
      Contact( "Liga_10" )
      Move(in := 16#0001, out1 => "Modbus_Send_Receive"."42028")
      wire#w1
      Contact( "Comm_ok" )
      { S7_Templates := "SrcType := Int" } EQ_Contact(in1 := "IEC_Counter_0_DB".CV, in2 := 99)
      I_Contact( "Modbus_Master_DB".BUSY )
   END_RUNG wire#w2
   RUNG wire#powerrail
      Contact( "Desliga_10" )
      Move(in := 16#0000, out1 => "Modbus_Send_Receive"."42028")
   END_RUNG wire#w1
   // the same network as SCL:
   IF "Liga_10" THEN "Modbus_Send_Receive"."42028" := 16#0001; END_IF;
   IF "Desliga_10" THEN "Modbus_Send_Receive"."42028" := 16#0000; END_IF;
   IF "IEC_Counter_0_DB".CV = 99 THEN
       "Modbus_Master_DB"(REQ := ("Liga_10" OR "Desliga_10") AND "Comm_ok" AND ("IEC_Counter_0_DB".CV = 99) AND NOT "Modbus_Master_DB".BUSY,   // Modbus_Master
                          MB_ADDR := 1,
                          MODE := 1,
                          DATA_ADDR := 42028,
                          DATA_LEN := 1,
                          DATA_PTR := "Modbus_Send_Receive"."42028",
                          DONE => "Modbus".Done,
                          BUSY => "Modbus".Busy,
                          ERROR => "Modbus".Error,
                          STATUS => "Modbus".Status);
   END_IF;
END_REGION

REGION Network 106: WR 42029 - OPER MODE
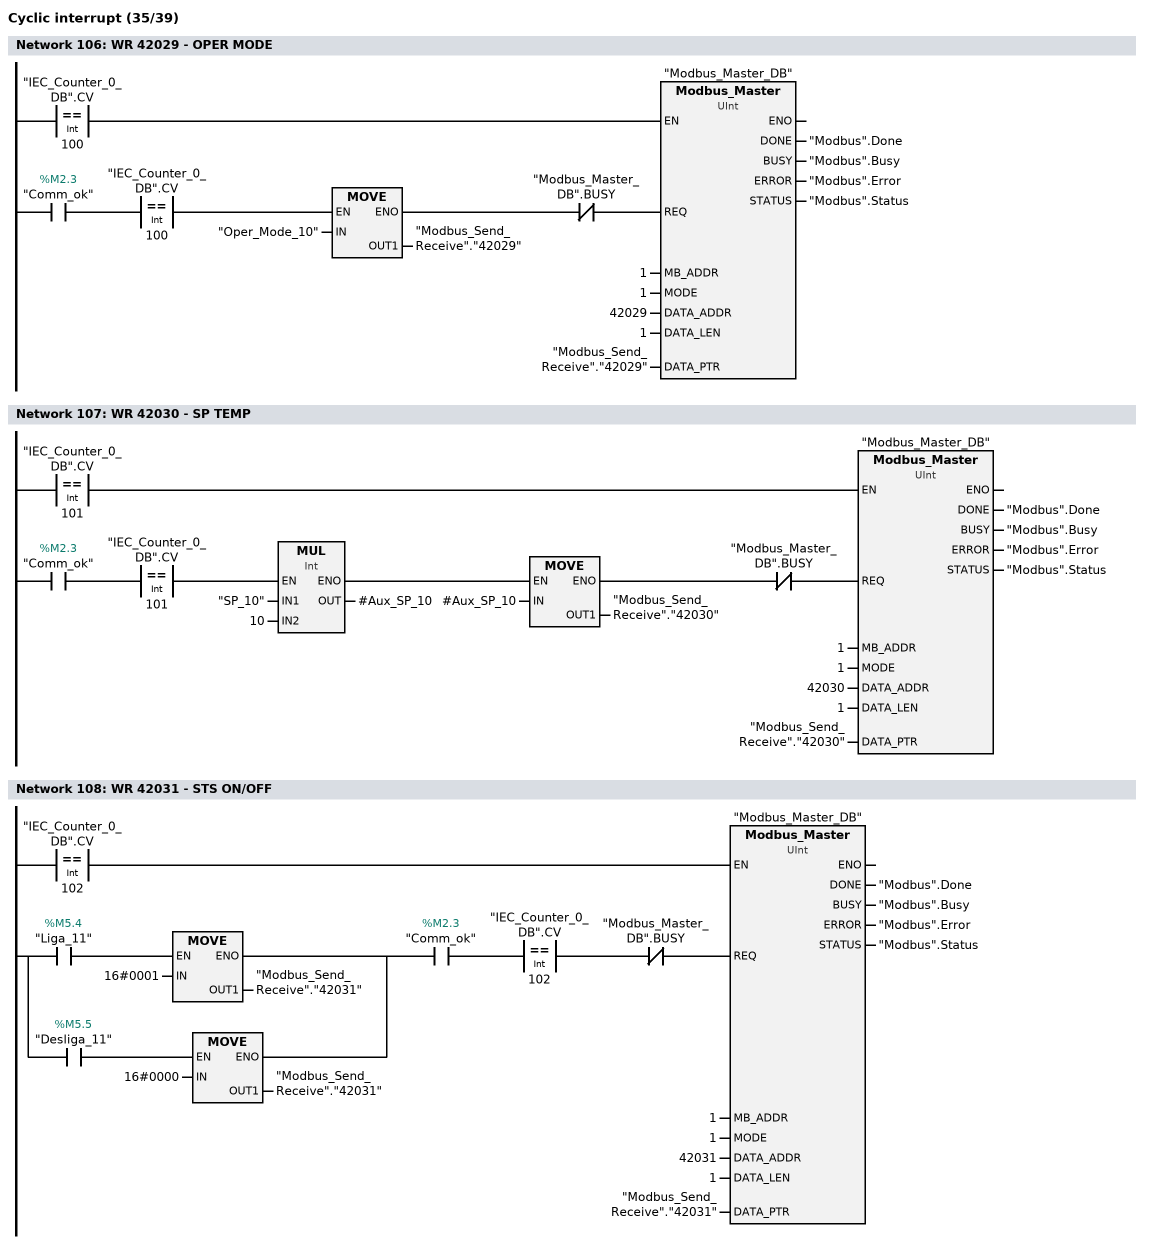
   RUNG wire#powerrail
      { S7_Templates := "SrcType := Int" } EQ_Contact(in1 := "IEC_Counter_0_DB".CV, in2 := 100)
      { S7_Templates := "[card := 0, word_type := UInt, dword_type := UDInt, byte_type := USInt, any_type := Variant]" } "Modbus_Master_DB".Modbus_Master(REQ := wire#w1, MB_ADDR := 1, MODE := 1, DATA_ADDR := 42029, DATA_LEN := 1, DATA_PTR := "Modbus_Send_Receive"."42029", DONE => "Modbus".Done, BUSY => "Modbus".Busy, ERROR => "Modbus".Error, STATUS => "Modbus".Status)
   END_RUNG
   RUNG wire#powerrail
      Contact( "Comm_ok" )
      { S7_Templates := "SrcType := Int" } EQ_Contact(in1 := "IEC_Counter_0_DB".CV, in2 := 100)
      Move(in := "Oper_Mode_10", out1 => "Modbus_Send_Receive"."42029")
      I_Contact( "Modbus_Master_DB".BUSY )
   END_RUNG wire#w1
   // the same network as SCL:
   #_w1 := "Comm_ok" AND ("IEC_Counter_0_DB".CV = 100);
   IF #_w1 THEN "Modbus_Send_Receive"."42029" := "Oper_Mode_10"; END_IF;
   IF "IEC_Counter_0_DB".CV = 100 THEN
       "Modbus_Master_DB"(REQ := #_w1 AND NOT "Modbus_Master_DB".BUSY,   // Modbus_Master
                          MB_ADDR := 1,
                          MODE := 1,
                          DATA_ADDR := 42029,
                          DATA_LEN := 1,
                          DATA_PTR := "Modbus_Send_Receive"."42029",
                          DONE => "Modbus".Done,
                          BUSY => "Modbus".Busy,
                          ERROR => "Modbus".Error,
                          STATUS => "Modbus".Status);
   END_IF;
END_REGION

REGION Network 107: WR 42030 - SP TEMP
   RUNG wire#powerrail
      { S7_Templates := "SrcType := Int" } EQ_Contact(in1 := "IEC_Counter_0_DB".CV, in2 := 101)
      { S7_Templates := "[card := 0, word_type := UInt, dword_type := UDInt, byte_type := USInt, any_type := Variant]" } "Modbus_Master_DB".Modbus_Master(REQ := wire#w1, MB_ADDR := 1, MODE := 1, DATA_ADDR := 42030, DATA_LEN := 1, DATA_PTR := "Modbus_Send_Receive"."42030", DONE => "Modbus".Done, BUSY => "Modbus".Busy, ERROR => "Modbus".Error, STATUS => "Modbus".Status)
   END_RUNG
   RUNG wire#powerrail
      Contact( "Comm_ok" )
      { S7_Templates := "SrcType := Int" } EQ_Contact(in1 := "IEC_Counter_0_DB".CV, in2 := 101)
      { S7_Templates := "SrcType := Int" } Mul(in1 := "SP_10", in2 := 10, out => #Aux_SP_10)
      Move(in := #Aux_SP_10, out1 => "Modbus_Send_Receive"."42030")
      I_Contact( "Modbus_Master_DB".BUSY )
   END_RUNG wire#w1
   // the same network as SCL:
   #_w1 := "Comm_ok" AND ("IEC_Counter_0_DB".CV = 101);
   IF #_w1 THEN
       #Aux_SP_10 := "SP_10" * 10;
       "Modbus_Send_Receive"."42030" := #Aux_SP_10;
   END_IF;
   IF "IEC_Counter_0_DB".CV = 101 THEN
       "Modbus_Master_DB"(REQ := #_w1 AND NOT "Modbus_Master_DB".BUSY,   // Modbus_Master
                          MB_ADDR := 1,
                          MODE := 1,
                          DATA_ADDR := 42030,
                          DATA_LEN := 1,
                          DATA_PTR := "Modbus_Send_Receive"."42030",
                          DONE => "Modbus".Done,
                          BUSY => "Modbus".Busy,
                          ERROR => "Modbus".Error,
                          STATUS => "Modbus".Status);
   END_IF;
END_REGION

REGION Network 108: WR 42031 - STS ON/OFF
   RUNG wire#powerrail
      { S7_Templates := "SrcType := Int" } EQ_Contact(in1 := "IEC_Counter_0_DB".CV, in2 := 102)
      { S7_Templates := "[card := 0, word_type := UInt, dword_type := UDInt, byte_type := USInt, any_type := Variant]" } "Modbus_Master_DB".Modbus_Master(REQ := wire#w2, MB_ADDR := 1, MODE := 1, DATA_ADDR := 42031, DATA_LEN := 1, DATA_PTR := "Modbus_Send_Receive"."42031", DONE => "Modbus".Done, BUSY => "Modbus".Busy, ERROR => "Modbus".Error, STATUS => "Modbus".Status)
   END_RUNG
   RUNG wire#powerrail
      Contact( "Liga_11" )
      Move(in := 16#0001, out1 => "Modbus_Send_Receive"."42031")
      wire#w1
      Contact( "Comm_ok" )
      { S7_Templates := "SrcType := Int" } EQ_Contact(in1 := "IEC_Counter_0_DB".CV, in2 := 102)
      I_Contact( "Modbus_Master_DB".BUSY )
   END_RUNG wire#w2
   RUNG wire#powerrail
      Contact( "Desliga_11" )
      Move(in := 16#0000, out1 => "Modbus_Send_Receive"."42031")
   END_RUNG wire#w1
   // the same network as SCL:
   IF "Liga_11" THEN "Modbus_Send_Receive"."42031" := 16#0001; END_IF;
   IF "Desliga_11" THEN "Modbus_Send_Receive"."42031" := 16#0000; END_IF;
   IF "IEC_Counter_0_DB".CV = 102 THEN
       "Modbus_Master_DB"(REQ := ("Liga_11" OR "Desliga_11") AND "Comm_ok" AND ("IEC_Counter_0_DB".CV = 102) AND NOT "Modbus_Master_DB".BUSY,   // Modbus_Master
                          MB_ADDR := 1,
                          MODE := 1,
                          DATA_ADDR := 42031,
                          DATA_LEN := 1,
                          DATA_PTR := "Modbus_Send_Receive"."42031",
                          DONE => "Modbus".Done,
                          BUSY => "Modbus".Busy,
                          ERROR => "Modbus".Error,
                          STATUS => "Modbus".Status);
   END_IF;
END_REGION

REGION Network 109: WR 42032 - OPER MODE
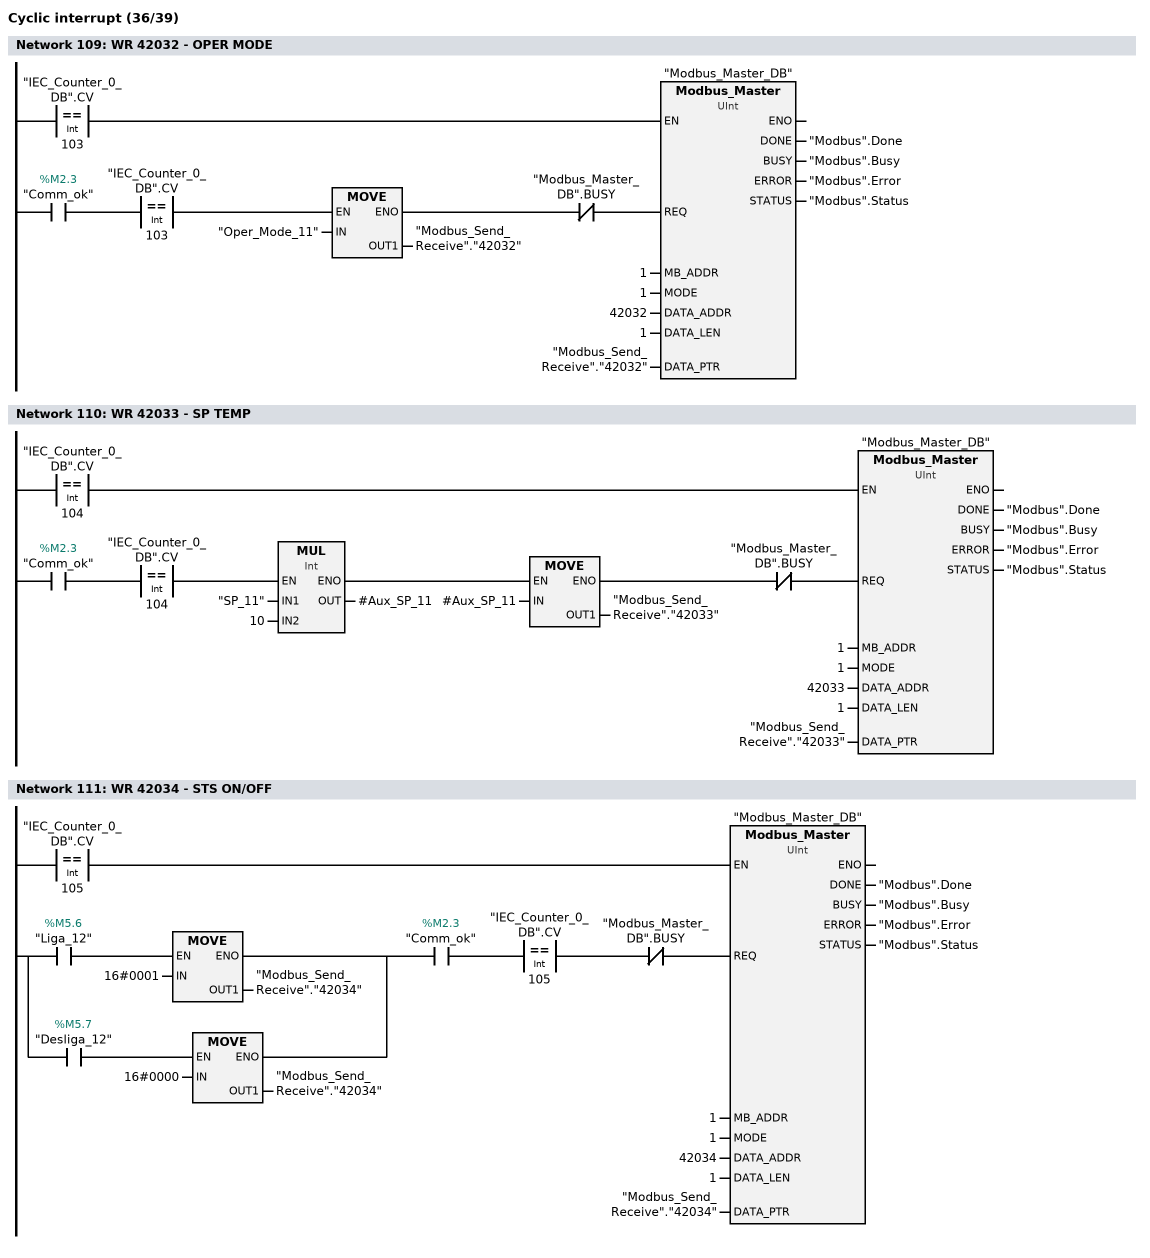
   RUNG wire#powerrail
      { S7_Templates := "SrcType := Int" } EQ_Contact(in1 := "IEC_Counter_0_DB".CV, in2 := 103)
      { S7_Templates := "[card := 0, word_type := UInt, dword_type := UDInt, byte_type := USInt, any_type := Variant]" } "Modbus_Master_DB".Modbus_Master(REQ := wire#w1, MB_ADDR := 1, MODE := 1, DATA_ADDR := 42032, DATA_LEN := 1, DATA_PTR := "Modbus_Send_Receive"."42032", DONE => "Modbus".Done, BUSY => "Modbus".Busy, ERROR => "Modbus".Error, STATUS => "Modbus".Status)
   END_RUNG
   RUNG wire#powerrail
      Contact( "Comm_ok" )
      { S7_Templates := "SrcType := Int" } EQ_Contact(in1 := "IEC_Counter_0_DB".CV, in2 := 103)
      Move(in := "Oper_Mode_11", out1 => "Modbus_Send_Receive"."42032")
      I_Contact( "Modbus_Master_DB".BUSY )
   END_RUNG wire#w1
   // the same network as SCL:
   #_w1 := "Comm_ok" AND ("IEC_Counter_0_DB".CV = 103);
   IF #_w1 THEN "Modbus_Send_Receive"."42032" := "Oper_Mode_11"; END_IF;
   IF "IEC_Counter_0_DB".CV = 103 THEN
       "Modbus_Master_DB"(REQ := #_w1 AND NOT "Modbus_Master_DB".BUSY,   // Modbus_Master
                          MB_ADDR := 1,
                          MODE := 1,
                          DATA_ADDR := 42032,
                          DATA_LEN := 1,
                          DATA_PTR := "Modbus_Send_Receive"."42032",
                          DONE => "Modbus".Done,
                          BUSY => "Modbus".Busy,
                          ERROR => "Modbus".Error,
                          STATUS => "Modbus".Status);
   END_IF;
END_REGION

REGION Network 110: WR 42033 - SP TEMP
   RUNG wire#powerrail
      { S7_Templates := "SrcType := Int" } EQ_Contact(in1 := "IEC_Counter_0_DB".CV, in2 := 104)
      { S7_Templates := "[card := 0, word_type := UInt, dword_type := UDInt, byte_type := USInt, any_type := Variant]" } "Modbus_Master_DB".Modbus_Master(REQ := wire#w1, MB_ADDR := 1, MODE := 1, DATA_ADDR := 42033, DATA_LEN := 1, DATA_PTR := "Modbus_Send_Receive"."42033", DONE => "Modbus".Done, BUSY => "Modbus".Busy, ERROR => "Modbus".Error, STATUS => "Modbus".Status)
   END_RUNG
   RUNG wire#powerrail
      Contact( "Comm_ok" )
      { S7_Templates := "SrcType := Int" } EQ_Contact(in1 := "IEC_Counter_0_DB".CV, in2 := 104)
      { S7_Templates := "SrcType := Int" } Mul(in1 := "SP_11", in2 := 10, out => #Aux_SP_11)
      Move(in := #Aux_SP_11, out1 => "Modbus_Send_Receive"."42033")
      I_Contact( "Modbus_Master_DB".BUSY )
   END_RUNG wire#w1
   // the same network as SCL:
   #_w1 := "Comm_ok" AND ("IEC_Counter_0_DB".CV = 104);
   IF #_w1 THEN
       #Aux_SP_11 := "SP_11" * 10;
       "Modbus_Send_Receive"."42033" := #Aux_SP_11;
   END_IF;
   IF "IEC_Counter_0_DB".CV = 104 THEN
       "Modbus_Master_DB"(REQ := #_w1 AND NOT "Modbus_Master_DB".BUSY,   // Modbus_Master
                          MB_ADDR := 1,
                          MODE := 1,
                          DATA_ADDR := 42033,
                          DATA_LEN := 1,
                          DATA_PTR := "Modbus_Send_Receive"."42033",
                          DONE => "Modbus".Done,
                          BUSY => "Modbus".Busy,
                          ERROR => "Modbus".Error,
                          STATUS => "Modbus".Status);
   END_IF;
END_REGION

REGION Network 111: WR 42034 - STS ON/OFF
   RUNG wire#powerrail
      { S7_Templates := "SrcType := Int" } EQ_Contact(in1 := "IEC_Counter_0_DB".CV, in2 := 105)
      { S7_Templates := "[card := 0, word_type := UInt, dword_type := UDInt, byte_type := USInt, any_type := Variant]" } "Modbus_Master_DB".Modbus_Master(REQ := wire#w2, MB_ADDR := 1, MODE := 1, DATA_ADDR := 42034, DATA_LEN := 1, DATA_PTR := "Modbus_Send_Receive"."42034", DONE => "Modbus".Done, BUSY => "Modbus".Busy, ERROR => "Modbus".Error, STATUS => "Modbus".Status)
   END_RUNG
   RUNG wire#powerrail
      Contact( "Liga_12" )
      Move(in := 16#0001, out1 => "Modbus_Send_Receive"."42034")
      wire#w1
      Contact( "Comm_ok" )
      { S7_Templates := "SrcType := Int" } EQ_Contact(in1 := "IEC_Counter_0_DB".CV, in2 := 105)
      I_Contact( "Modbus_Master_DB".BUSY )
   END_RUNG wire#w2
   RUNG wire#powerrail
      Contact( "Desliga_12" )
      Move(in := 16#0000, out1 => "Modbus_Send_Receive"."42034")
   END_RUNG wire#w1
   // the same network as SCL:
   IF "Liga_12" THEN "Modbus_Send_Receive"."42034" := 16#0001; END_IF;
   IF "Desliga_12" THEN "Modbus_Send_Receive"."42034" := 16#0000; END_IF;
   IF "IEC_Counter_0_DB".CV = 105 THEN
       "Modbus_Master_DB"(REQ := ("Liga_12" OR "Desliga_12") AND "Comm_ok" AND ("IEC_Counter_0_DB".CV = 105) AND NOT "Modbus_Master_DB".BUSY,   // Modbus_Master
                          MB_ADDR := 1,
                          MODE := 1,
                          DATA_ADDR := 42034,
                          DATA_LEN := 1,
                          DATA_PTR := "Modbus_Send_Receive"."42034",
                          DONE => "Modbus".Done,
                          BUSY => "Modbus".Busy,
                          ERROR => "Modbus".Error,
                          STATUS => "Modbus".Status);
   END_IF;
END_REGION

REGION Network 112: WR 42035 - OPER MODE
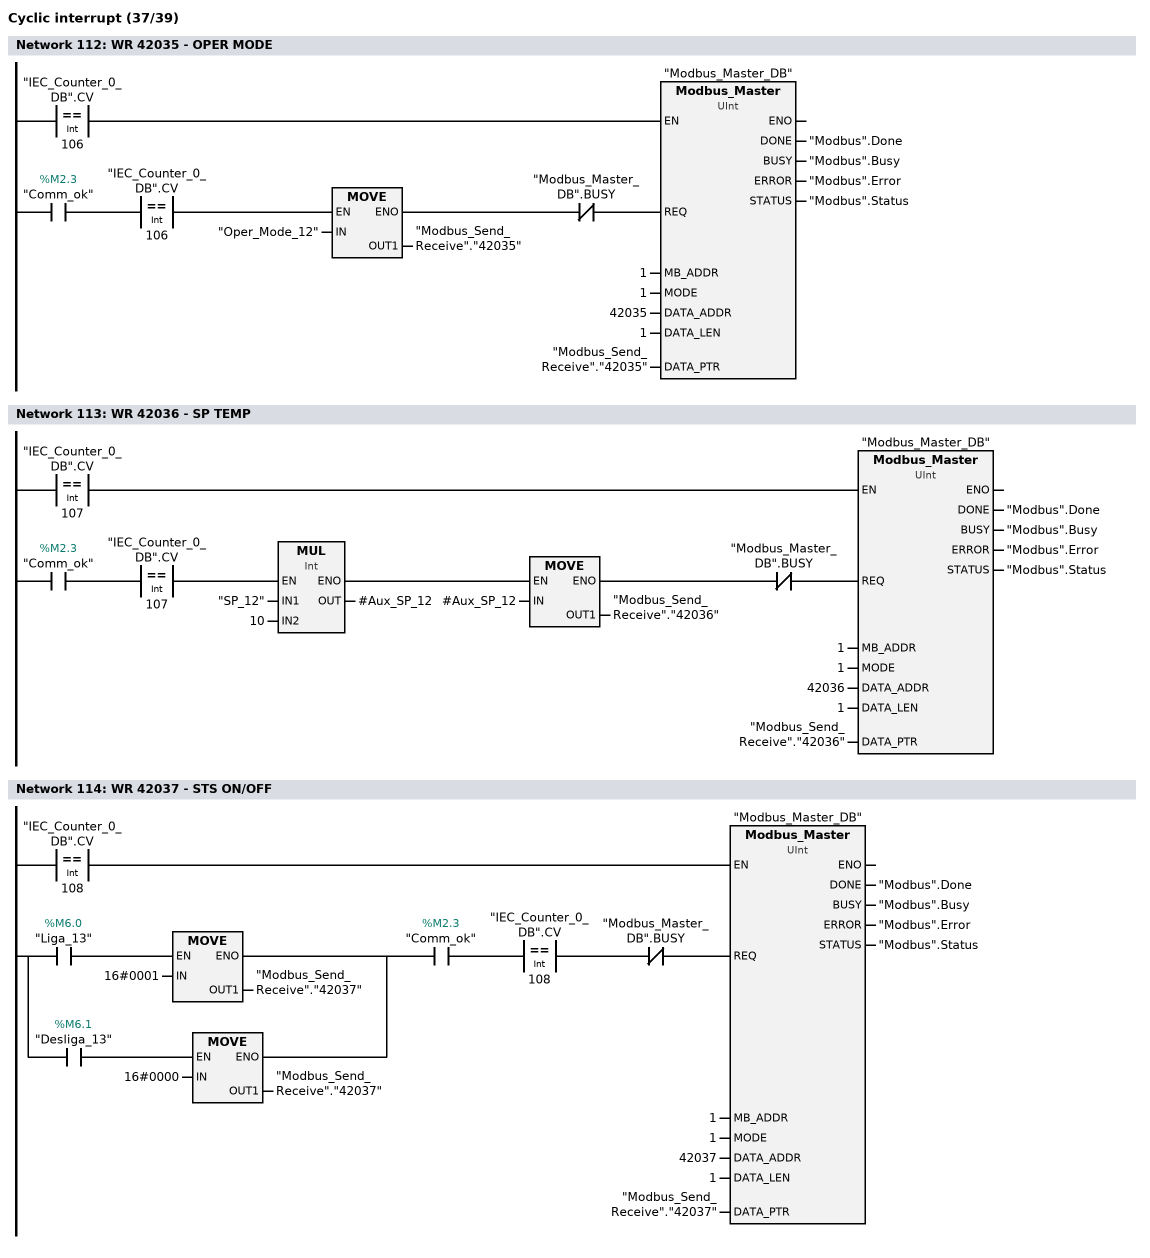
   RUNG wire#powerrail
      { S7_Templates := "SrcType := Int" } EQ_Contact(in1 := "IEC_Counter_0_DB".CV, in2 := 106)
      { S7_Templates := "[card := 0, word_type := UInt, dword_type := UDInt, byte_type := USInt, any_type := Variant]" } "Modbus_Master_DB".Modbus_Master(REQ := wire#w1, MB_ADDR := 1, MODE := 1, DATA_ADDR := 42035, DATA_LEN := 1, DATA_PTR := "Modbus_Send_Receive"."42035", DONE => "Modbus".Done, BUSY => "Modbus".Busy, ERROR => "Modbus".Error, STATUS => "Modbus".Status)
   END_RUNG
   RUNG wire#powerrail
      Contact( "Comm_ok" )
      { S7_Templates := "SrcType := Int" } EQ_Contact(in1 := "IEC_Counter_0_DB".CV, in2 := 106)
      Move(in := "Oper_Mode_12", out1 => "Modbus_Send_Receive"."42035")
      I_Contact( "Modbus_Master_DB".BUSY )
   END_RUNG wire#w1
   // the same network as SCL:
   #_w1 := "Comm_ok" AND ("IEC_Counter_0_DB".CV = 106);
   IF #_w1 THEN "Modbus_Send_Receive"."42035" := "Oper_Mode_12"; END_IF;
   IF "IEC_Counter_0_DB".CV = 106 THEN
       "Modbus_Master_DB"(REQ := #_w1 AND NOT "Modbus_Master_DB".BUSY,   // Modbus_Master
                          MB_ADDR := 1,
                          MODE := 1,
                          DATA_ADDR := 42035,
                          DATA_LEN := 1,
                          DATA_PTR := "Modbus_Send_Receive"."42035",
                          DONE => "Modbus".Done,
                          BUSY => "Modbus".Busy,
                          ERROR => "Modbus".Error,
                          STATUS => "Modbus".Status);
   END_IF;
END_REGION

REGION Network 113: WR 42036 - SP TEMP
   RUNG wire#powerrail
      { S7_Templates := "SrcType := Int" } EQ_Contact(in1 := "IEC_Counter_0_DB".CV, in2 := 107)
      { S7_Templates := "[card := 0, word_type := UInt, dword_type := UDInt, byte_type := USInt, any_type := Variant]" } "Modbus_Master_DB".Modbus_Master(REQ := wire#w1, MB_ADDR := 1, MODE := 1, DATA_ADDR := 42036, DATA_LEN := 1, DATA_PTR := "Modbus_Send_Receive"."42036", DONE => "Modbus".Done, BUSY => "Modbus".Busy, ERROR => "Modbus".Error, STATUS => "Modbus".Status)
   END_RUNG
   RUNG wire#powerrail
      Contact( "Comm_ok" )
      { S7_Templates := "SrcType := Int" } EQ_Contact(in1 := "IEC_Counter_0_DB".CV, in2 := 107)
      { S7_Templates := "SrcType := Int" } Mul(in1 := "SP_12", in2 := 10, out => #Aux_SP_12)
      Move(in := #Aux_SP_12, out1 => "Modbus_Send_Receive"."42036")
      I_Contact( "Modbus_Master_DB".BUSY )
   END_RUNG wire#w1
   // the same network as SCL:
   #_w1 := "Comm_ok" AND ("IEC_Counter_0_DB".CV = 107);
   IF #_w1 THEN
       #Aux_SP_12 := "SP_12" * 10;
       "Modbus_Send_Receive"."42036" := #Aux_SP_12;
   END_IF;
   IF "IEC_Counter_0_DB".CV = 107 THEN
       "Modbus_Master_DB"(REQ := #_w1 AND NOT "Modbus_Master_DB".BUSY,   // Modbus_Master
                          MB_ADDR := 1,
                          MODE := 1,
                          DATA_ADDR := 42036,
                          DATA_LEN := 1,
                          DATA_PTR := "Modbus_Send_Receive"."42036",
                          DONE => "Modbus".Done,
                          BUSY => "Modbus".Busy,
                          ERROR => "Modbus".Error,
                          STATUS => "Modbus".Status);
   END_IF;
END_REGION

REGION Network 114: WR 42037 - STS ON/OFF
   RUNG wire#powerrail
      { S7_Templates := "SrcType := Int" } EQ_Contact(in1 := "IEC_Counter_0_DB".CV, in2 := 108)
      { S7_Templates := "[card := 0, word_type := UInt, dword_type := UDInt, byte_type := USInt, any_type := Variant]" } "Modbus_Master_DB".Modbus_Master(REQ := wire#w2, MB_ADDR := 1, MODE := 1, DATA_ADDR := 42037, DATA_LEN := 1, DATA_PTR := "Modbus_Send_Receive"."42037", DONE => "Modbus".Done, BUSY => "Modbus".Busy, ERROR => "Modbus".Error, STATUS => "Modbus".Status)
   END_RUNG
   RUNG wire#powerrail
      Contact( "Liga_13" )
      Move(in := 16#0001, out1 => "Modbus_Send_Receive"."42037")
      wire#w1
      Contact( "Comm_ok" )
      { S7_Templates := "SrcType := Int" } EQ_Contact(in1 := "IEC_Counter_0_DB".CV, in2 := 108)
      I_Contact( "Modbus_Master_DB".BUSY )
   END_RUNG wire#w2
   RUNG wire#powerrail
      Contact( "Desliga_13" )
      Move(in := 16#0000, out1 => "Modbus_Send_Receive"."42037")
   END_RUNG wire#w1
   // the same network as SCL:
   IF "Liga_13" THEN "Modbus_Send_Receive"."42037" := 16#0001; END_IF;
   IF "Desliga_13" THEN "Modbus_Send_Receive"."42037" := 16#0000; END_IF;
   IF "IEC_Counter_0_DB".CV = 108 THEN
       "Modbus_Master_DB"(REQ := ("Liga_13" OR "Desliga_13") AND "Comm_ok" AND ("IEC_Counter_0_DB".CV = 108) AND NOT "Modbus_Master_DB".BUSY,   // Modbus_Master
                          MB_ADDR := 1,
                          MODE := 1,
                          DATA_ADDR := 42037,
                          DATA_LEN := 1,
                          DATA_PTR := "Modbus_Send_Receive"."42037",
                          DONE => "Modbus".Done,
                          BUSY => "Modbus".Busy,
                          ERROR => "Modbus".Error,
                          STATUS => "Modbus".Status);
   END_IF;
END_REGION

REGION Network 115: WR 42038 - OPER MODE
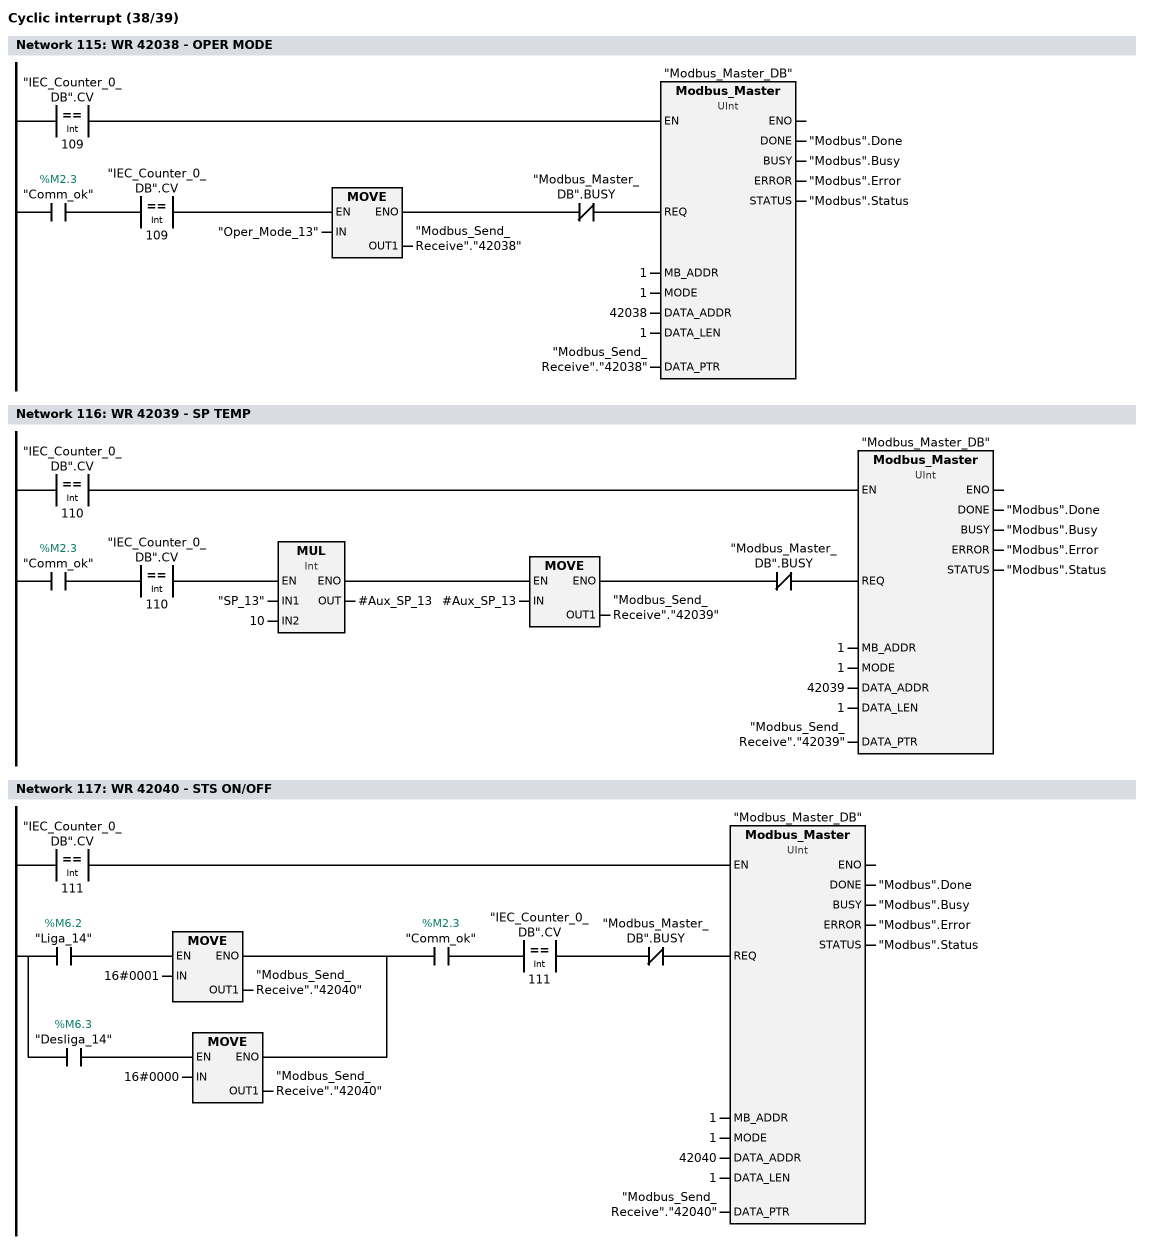
   RUNG wire#powerrail
      { S7_Templates := "SrcType := Int" } EQ_Contact(in1 := "IEC_Counter_0_DB".CV, in2 := 109)
      { S7_Templates := "[card := 0, word_type := UInt, dword_type := UDInt, byte_type := USInt, any_type := Variant]" } "Modbus_Master_DB".Modbus_Master(REQ := wire#w1, MB_ADDR := 1, MODE := 1, DATA_ADDR := 42038, DATA_LEN := 1, DATA_PTR := "Modbus_Send_Receive"."42038", DONE => "Modbus".Done, BUSY => "Modbus".Busy, ERROR => "Modbus".Error, STATUS => "Modbus".Status)
   END_RUNG
   RUNG wire#powerrail
      Contact( "Comm_ok" )
      { S7_Templates := "SrcType := Int" } EQ_Contact(in1 := "IEC_Counter_0_DB".CV, in2 := 109)
      Move(in := "Oper_Mode_13", out1 => "Modbus_Send_Receive"."42038")
      I_Contact( "Modbus_Master_DB".BUSY )
   END_RUNG wire#w1
   // the same network as SCL:
   #_w1 := "Comm_ok" AND ("IEC_Counter_0_DB".CV = 109);
   IF #_w1 THEN "Modbus_Send_Receive"."42038" := "Oper_Mode_13"; END_IF;
   IF "IEC_Counter_0_DB".CV = 109 THEN
       "Modbus_Master_DB"(REQ := #_w1 AND NOT "Modbus_Master_DB".BUSY,   // Modbus_Master
                          MB_ADDR := 1,
                          MODE := 1,
                          DATA_ADDR := 42038,
                          DATA_LEN := 1,
                          DATA_PTR := "Modbus_Send_Receive"."42038",
                          DONE => "Modbus".Done,
                          BUSY => "Modbus".Busy,
                          ERROR => "Modbus".Error,
                          STATUS => "Modbus".Status);
   END_IF;
END_REGION

REGION Network 116: WR 42039 - SP TEMP
   RUNG wire#powerrail
      { S7_Templates := "SrcType := Int" } EQ_Contact(in1 := "IEC_Counter_0_DB".CV, in2 := 110)
      { S7_Templates := "[card := 0, word_type := UInt, dword_type := UDInt, byte_type := USInt, any_type := Variant]" } "Modbus_Master_DB".Modbus_Master(REQ := wire#w1, MB_ADDR := 1, MODE := 1, DATA_ADDR := 42039, DATA_LEN := 1, DATA_PTR := "Modbus_Send_Receive"."42039", DONE => "Modbus".Done, BUSY => "Modbus".Busy, ERROR => "Modbus".Error, STATUS => "Modbus".Status)
   END_RUNG
   RUNG wire#powerrail
      Contact( "Comm_ok" )
      { S7_Templates := "SrcType := Int" } EQ_Contact(in1 := "IEC_Counter_0_DB".CV, in2 := 110)
      { S7_Templates := "SrcType := Int" } Mul(in1 := "SP_13", in2 := 10, out => #Aux_SP_13)
      Move(in := #Aux_SP_13, out1 => "Modbus_Send_Receive"."42039")
      I_Contact( "Modbus_Master_DB".BUSY )
   END_RUNG wire#w1
   // the same network as SCL:
   #_w1 := "Comm_ok" AND ("IEC_Counter_0_DB".CV = 110);
   IF #_w1 THEN
       #Aux_SP_13 := "SP_13" * 10;
       "Modbus_Send_Receive"."42039" := #Aux_SP_13;
   END_IF;
   IF "IEC_Counter_0_DB".CV = 110 THEN
       "Modbus_Master_DB"(REQ := #_w1 AND NOT "Modbus_Master_DB".BUSY,   // Modbus_Master
                          MB_ADDR := 1,
                          MODE := 1,
                          DATA_ADDR := 42039,
                          DATA_LEN := 1,
                          DATA_PTR := "Modbus_Send_Receive"."42039",
                          DONE => "Modbus".Done,
                          BUSY => "Modbus".Busy,
                          ERROR => "Modbus".Error,
                          STATUS => "Modbus".Status);
   END_IF;
END_REGION

REGION Network 117: WR 42040 - STS ON/OFF
   RUNG wire#powerrail
      { S7_Templates := "SrcType := Int" } EQ_Contact(in1 := "IEC_Counter_0_DB".CV, in2 := 111)
      { S7_Templates := "[card := 0, word_type := UInt, dword_type := UDInt, byte_type := USInt, any_type := Variant]" } "Modbus_Master_DB".Modbus_Master(REQ := wire#w2, MB_ADDR := 1, MODE := 1, DATA_ADDR := 42040, DATA_LEN := 1, DATA_PTR := "Modbus_Send_Receive"."42040", DONE => "Modbus".Done, BUSY => "Modbus".Busy, ERROR => "Modbus".Error, STATUS => "Modbus".Status)
   END_RUNG
   RUNG wire#powerrail
      Contact( "Liga_14" )
      Move(in := 16#0001, out1 => "Modbus_Send_Receive"."42040")
      wire#w1
      Contact( "Comm_ok" )
      { S7_Templates := "SrcType := Int" } EQ_Contact(in1 := "IEC_Counter_0_DB".CV, in2 := 111)
      I_Contact( "Modbus_Master_DB".BUSY )
   END_RUNG wire#w2
   RUNG wire#powerrail
      Contact( "Desliga_14" )
      Move(in := 16#0000, out1 => "Modbus_Send_Receive"."42040")
   END_RUNG wire#w1
   // the same network as SCL:
   IF "Liga_14" THEN "Modbus_Send_Receive"."42040" := 16#0001; END_IF;
   IF "Desliga_14" THEN "Modbus_Send_Receive"."42040" := 16#0000; END_IF;
   IF "IEC_Counter_0_DB".CV = 111 THEN
       "Modbus_Master_DB"(REQ := ("Liga_14" OR "Desliga_14") AND "Comm_ok" AND ("IEC_Counter_0_DB".CV = 111) AND NOT "Modbus_Master_DB".BUSY,   // Modbus_Master
                          MB_ADDR := 1,
                          MODE := 1,
                          DATA_ADDR := 42040,
                          DATA_LEN := 1,
                          DATA_PTR := "Modbus_Send_Receive"."42040",
                          DONE => "Modbus".Done,
                          BUSY => "Modbus".Busy,
                          ERROR => "Modbus".Error,
                          STATUS => "Modbus".Status);
   END_IF;
END_REGION

REGION Network 118: WR 42041 - OPER MODE
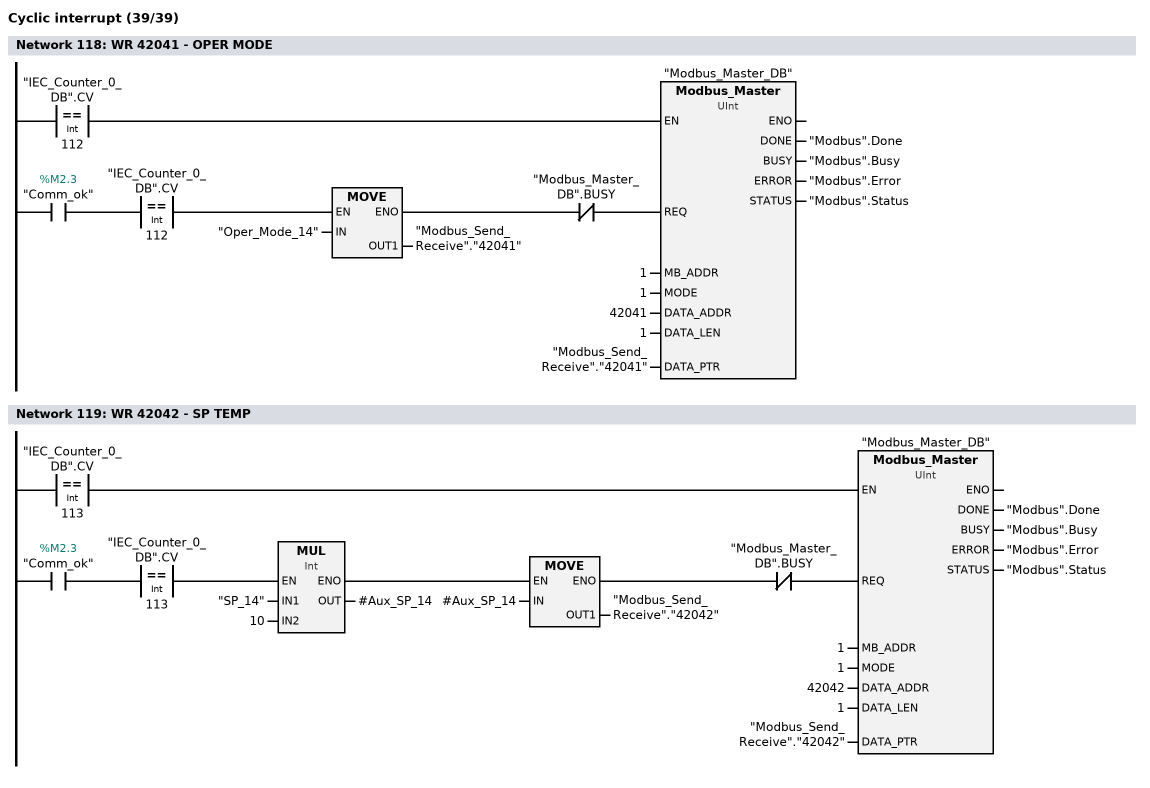
   RUNG wire#powerrail
      { S7_Templates := "SrcType := Int" } EQ_Contact(in1 := "IEC_Counter_0_DB".CV, in2 := 112)
      { S7_Templates := "[card := 0, word_type := UInt, dword_type := UDInt, byte_type := USInt, any_type := Variant]" } "Modbus_Master_DB".Modbus_Master(REQ := wire#w1, MB_ADDR := 1, MODE := 1, DATA_ADDR := 42041, DATA_LEN := 1, DATA_PTR := "Modbus_Send_Receive"."42041", DONE => "Modbus".Done, BUSY => "Modbus".Busy, ERROR => "Modbus".Error, STATUS => "Modbus".Status)
   END_RUNG
   RUNG wire#powerrail
      Contact( "Comm_ok" )
      { S7_Templates := "SrcType := Int" } EQ_Contact(in1 := "IEC_Counter_0_DB".CV, in2 := 112)
      Move(in := "Oper_Mode_14", out1 => "Modbus_Send_Receive"."42041")
      I_Contact( "Modbus_Master_DB".BUSY )
   END_RUNG wire#w1
   // the same network as SCL:
   #_w1 := "Comm_ok" AND ("IEC_Counter_0_DB".CV = 112);
   IF #_w1 THEN "Modbus_Send_Receive"."42041" := "Oper_Mode_14"; END_IF;
   IF "IEC_Counter_0_DB".CV = 112 THEN
       "Modbus_Master_DB"(REQ := #_w1 AND NOT "Modbus_Master_DB".BUSY,   // Modbus_Master
                          MB_ADDR := 1,
                          MODE := 1,
                          DATA_ADDR := 42041,
                          DATA_LEN := 1,
                          DATA_PTR := "Modbus_Send_Receive"."42041",
                          DONE => "Modbus".Done,
                          BUSY => "Modbus".Busy,
                          ERROR => "Modbus".Error,
                          STATUS => "Modbus".Status);
   END_IF;
END_REGION

REGION Network 119: WR 42042 - SP TEMP
   RUNG wire#powerrail
      { S7_Templates := "SrcType := Int" } EQ_Contact(in1 := "IEC_Counter_0_DB".CV, in2 := 113)
      { S7_Templates := "[card := 0, word_type := UInt, dword_type := UDInt, byte_type := USInt, any_type := Variant]" } "Modbus_Master_DB".Modbus_Master(REQ := wire#w1, MB_ADDR := 1, MODE := 1, DATA_ADDR := 42042, DATA_LEN := 1, DATA_PTR := "Modbus_Send_Receive"."42042", DONE => "Modbus".Done, BUSY => "Modbus".Busy, ERROR => "Modbus".Error, STATUS => "Modbus".Status)
   END_RUNG
   RUNG wire#powerrail
      Contact( "Comm_ok" )
      { S7_Templates := "SrcType := Int" } EQ_Contact(in1 := "IEC_Counter_0_DB".CV, in2 := 113)
      { S7_Templates := "SrcType := Int" } Mul(in1 := "SP_14", in2 := 10, out => #Aux_SP_14)
      Move(in := #Aux_SP_14, out1 => "Modbus_Send_Receive"."42042")
      I_Contact( "Modbus_Master_DB".BUSY )
   END_RUNG wire#w1
   // the same network as SCL:
   #_w1 := "Comm_ok" AND ("IEC_Counter_0_DB".CV = 113);
   IF #_w1 THEN
       #Aux_SP_14 := "SP_14" * 10;
       "Modbus_Send_Receive"."42042" := #Aux_SP_14;
   END_IF;
   IF "IEC_Counter_0_DB".CV = 113 THEN
       "Modbus_Master_DB"(REQ := #_w1 AND NOT "Modbus_Master_DB".BUSY,   // Modbus_Master
                          MB_ADDR := 1,
                          MODE := 1,
                          DATA_ADDR := 42042,
                          DATA_LEN := 1,
                          DATA_PTR := "Modbus_Send_Receive"."42042",
                          DONE => "Modbus".Done,
                          BUSY => "Modbus".Busy,
                          ERROR => "Modbus".Error,
                          STATUS => "Modbus".Status);
   END_IF;
END_REGION
END_ORGANIZATION_BLOCK

FUNCTION "Sts_Auto_Manual" : Void   // FC3, LAD
{ S7_Optimized_Access := 'TRUE' }
VERSION : 0.1
// stored: AutoNumber true, IsIECCheckEnabled false, SetENOAutomatically false, UDAEnableTagReadback false
   VAR_INPUT
      "30001" : Word;
   END_VAR
   VAR_TEMP
      Aux_1 : Word;
   END_VAR
BEGIN

REGION Network 1
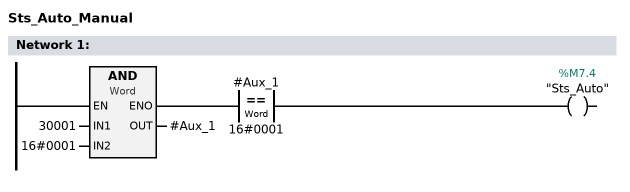
   RUNG wire#powerrail
      { S7_Templates := "SrcType := Word" } And(in1 := 30001, in2 := 16#0001, out => #Aux_1)
      { S7_Templates := "SrcType := Word" } EQ_Contact(in1 := #Aux_1, in2 := 16#0001)
      Coil( "Sts_Auto" )
   END_RUNG
   // the same network as SCL:
   #Aux_1 := 30001 AND 16#0001;
   "Sts_Auto" := #Aux_1 = 16#0001;
END_REGION
END_FUNCTION

FUNCTION "Data_Treatment" : Void   // FC2, LAD
{ S7_Optimized_Access := 'TRUE' }
VERSION : 0.1
// stored: AutoNumber true, IsIECCheckEnabled false, SetENOAutomatically false, UDAEnableTagReadback false
BEGIN

REGION Network 1: Extrusora 1
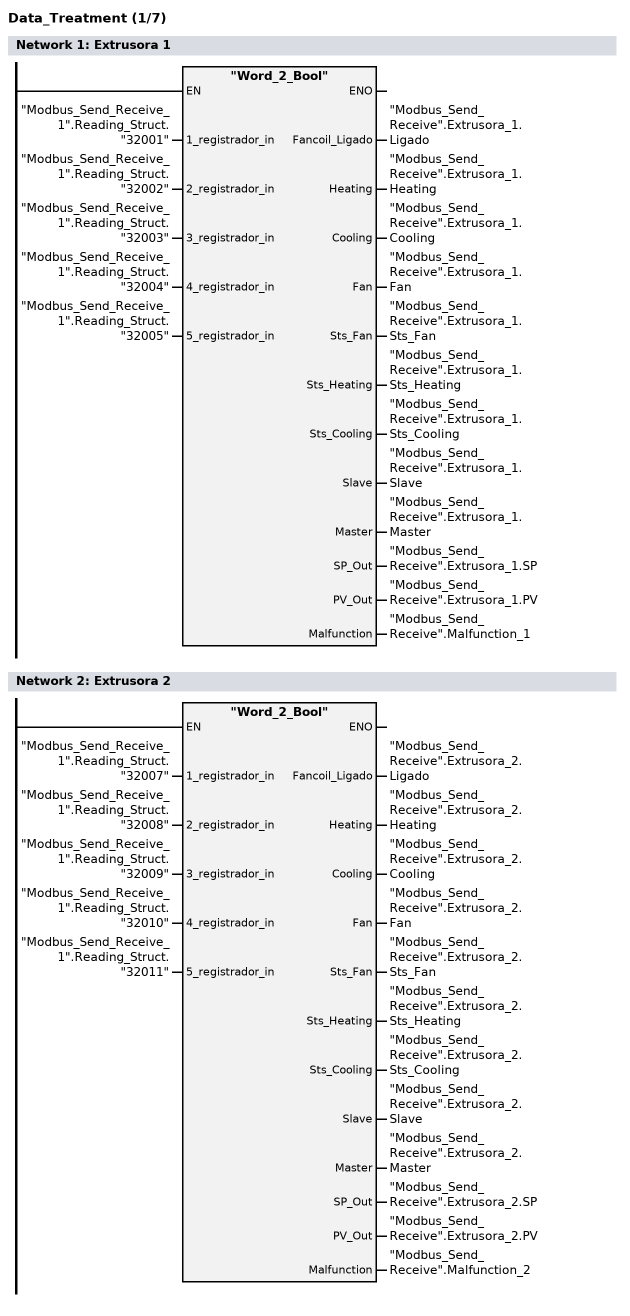
   RUNG wire#powerrail
      "Word_2_Bool"("1_registrador_in" := "Modbus_Send_Receive_1".Reading_Struct."32001", "2_registrador_in" := "Modbus_Send_Receive_1".Reading_Struct."32002", "3_registrador_in" := "Modbus_Send_Receive_1".Reading_Struct."32003", "4_registrador_in" := "Modbus_Send_Receive_1".Reading_Struct."32004", "5_registrador_in" := "Modbus_Send_Receive_1".Reading_Struct."32005", Fancoil_Ligado => "Modbus_Send_Receive".Extrusora_1.Ligado, Heating => "Modbus_Send_Receive".Extrusora_1.Heating, Cooling => "Modbus_Send_Receive".Extrusora_1.Cooling, Fan => "Modbus_Send_Receive".Extrusora_1.Fan, Sts_Fan => "Modbus_Send_Receive".Extrusora_1.Sts_Fan, Sts_Heating => "Modbus_Send_Receive".Extrusora_1.Sts_Heating, Sts_Cooling => "Modbus_Send_Receive".Extrusora_1.Sts_Cooling, Slave => "Modbus_Send_Receive".Extrusora_1.Slave, Master => "Modbus_Send_Receive".Extrusora_1.Master, SP_Out => "Modbus_Send_Receive".Extrusora_1.SP, PV_Out => "Modbus_Send_Receive".Extrusora_1.PV, Malfunction => "Modbus_Send_Receive".Malfunction_1)
   END_RUNG
   // the same network as SCL:
   "Word_2_Bool"("1_registrador_in" := "Modbus_Send_Receive_1".Reading_Struct."32001",
                 "2_registrador_in" := "Modbus_Send_Receive_1".Reading_Struct."32002",
                 "3_registrador_in" := "Modbus_Send_Receive_1".Reading_Struct."32003",
                 "4_registrador_in" := "Modbus_Send_Receive_1".Reading_Struct."32004",
                 "5_registrador_in" := "Modbus_Send_Receive_1".Reading_Struct."32005",
                 Fancoil_Ligado => "Modbus_Send_Receive".Extrusora_1.Ligado,
                 Heating => "Modbus_Send_Receive".Extrusora_1.Heating,
                 Cooling => "Modbus_Send_Receive".Extrusora_1.Cooling,
                 Fan => "Modbus_Send_Receive".Extrusora_1.Fan,
                 Sts_Fan => "Modbus_Send_Receive".Extrusora_1.Sts_Fan,
                 Sts_Heating => "Modbus_Send_Receive".Extrusora_1.Sts_Heating,
                 Sts_Cooling => "Modbus_Send_Receive".Extrusora_1.Sts_Cooling,
                 Slave => "Modbus_Send_Receive".Extrusora_1.Slave,
                 Master => "Modbus_Send_Receive".Extrusora_1.Master,
                 SP_Out => "Modbus_Send_Receive".Extrusora_1.SP,
                 PV_Out => "Modbus_Send_Receive".Extrusora_1.PV,
                 Malfunction => "Modbus_Send_Receive".Malfunction_1);
END_REGION

REGION Network 2: Extrusora 2
   RUNG wire#powerrail
      "Word_2_Bool"("1_registrador_in" := "Modbus_Send_Receive_1".Reading_Struct."32007", "2_registrador_in" := "Modbus_Send_Receive_1".Reading_Struct."32008", "3_registrador_in" := "Modbus_Send_Receive_1".Reading_Struct."32009", "4_registrador_in" := "Modbus_Send_Receive_1".Reading_Struct."32010", "5_registrador_in" := "Modbus_Send_Receive_1".Reading_Struct."32011", Fancoil_Ligado => "Modbus_Send_Receive".Extrusora_2.Ligado, Heating => "Modbus_Send_Receive".Extrusora_2.Heating, Cooling => "Modbus_Send_Receive".Extrusora_2.Cooling, Fan => "Modbus_Send_Receive".Extrusora_2.Fan, Sts_Fan => "Modbus_Send_Receive".Extrusora_2.Sts_Fan, Sts_Heating => "Modbus_Send_Receive".Extrusora_2.Sts_Heating, Sts_Cooling => "Modbus_Send_Receive".Extrusora_2.Sts_Cooling, Slave => "Modbus_Send_Receive".Extrusora_2.Slave, Master => "Modbus_Send_Receive".Extrusora_2.Master, SP_Out => "Modbus_Send_Receive".Extrusora_2.SP, PV_Out => "Modbus_Send_Receive".Extrusora_2.PV, Malfunction => "Modbus_Send_Receive".Malfunction_2)
   END_RUNG
   // the same network as SCL:
   "Word_2_Bool"("1_registrador_in" := "Modbus_Send_Receive_1".Reading_Struct."32007",
                 "2_registrador_in" := "Modbus_Send_Receive_1".Reading_Struct."32008",
                 "3_registrador_in" := "Modbus_Send_Receive_1".Reading_Struct."32009",
                 "4_registrador_in" := "Modbus_Send_Receive_1".Reading_Struct."32010",
                 "5_registrador_in" := "Modbus_Send_Receive_1".Reading_Struct."32011",
                 Fancoil_Ligado => "Modbus_Send_Receive".Extrusora_2.Ligado,
                 Heating => "Modbus_Send_Receive".Extrusora_2.Heating,
                 Cooling => "Modbus_Send_Receive".Extrusora_2.Cooling,
                 Fan => "Modbus_Send_Receive".Extrusora_2.Fan,
                 Sts_Fan => "Modbus_Send_Receive".Extrusora_2.Sts_Fan,
                 Sts_Heating => "Modbus_Send_Receive".Extrusora_2.Sts_Heating,
                 Sts_Cooling => "Modbus_Send_Receive".Extrusora_2.Sts_Cooling,
                 Slave => "Modbus_Send_Receive".Extrusora_2.Slave,
                 Master => "Modbus_Send_Receive".Extrusora_2.Master,
                 SP_Out => "Modbus_Send_Receive".Extrusora_2.SP,
                 PV_Out => "Modbus_Send_Receive".Extrusora_2.PV,
                 Malfunction => "Modbus_Send_Receive".Malfunction_2);
END_REGION

REGION Network 3: Extrusora 3
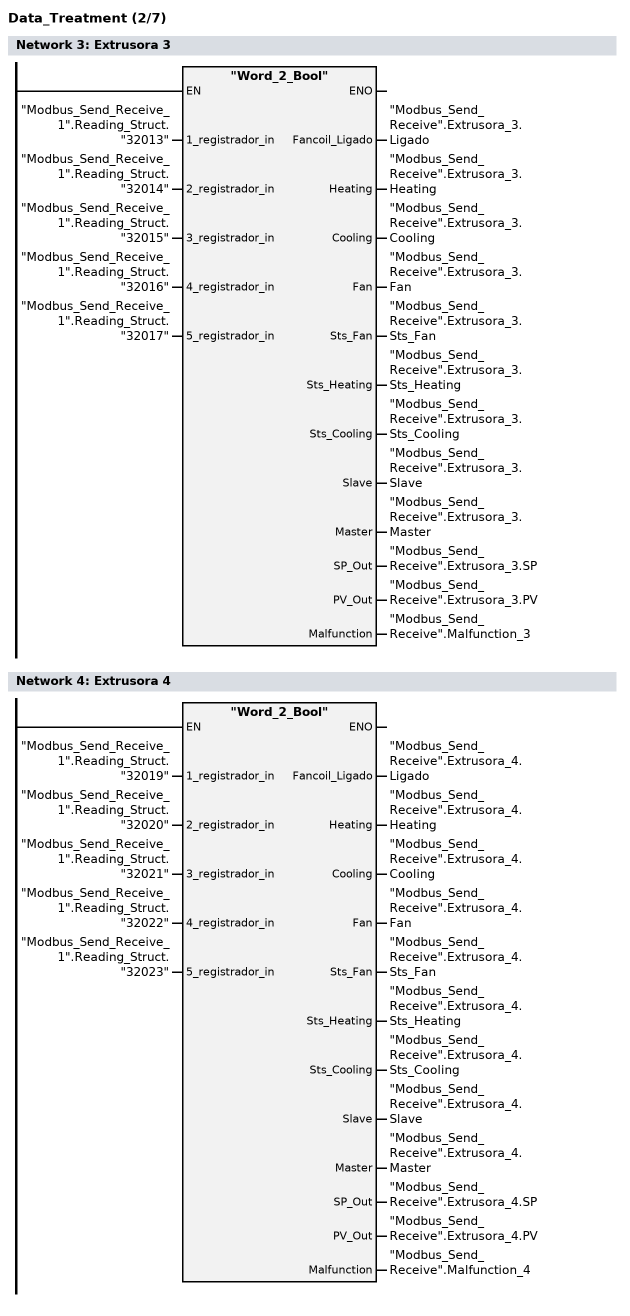
   RUNG wire#powerrail
      "Word_2_Bool"("1_registrador_in" := "Modbus_Send_Receive_1".Reading_Struct."32013", "2_registrador_in" := "Modbus_Send_Receive_1".Reading_Struct."32014", "3_registrador_in" := "Modbus_Send_Receive_1".Reading_Struct."32015", "4_registrador_in" := "Modbus_Send_Receive_1".Reading_Struct."32016", "5_registrador_in" := "Modbus_Send_Receive_1".Reading_Struct."32017", Fancoil_Ligado => "Modbus_Send_Receive".Extrusora_3.Ligado, Heating => "Modbus_Send_Receive".Extrusora_3.Heating, Cooling => "Modbus_Send_Receive".Extrusora_3.Cooling, Fan => "Modbus_Send_Receive".Extrusora_3.Fan, Sts_Fan => "Modbus_Send_Receive".Extrusora_3.Sts_Fan, Sts_Heating => "Modbus_Send_Receive".Extrusora_3.Sts_Heating, Sts_Cooling => "Modbus_Send_Receive".Extrusora_3.Sts_Cooling, Slave => "Modbus_Send_Receive".Extrusora_3.Slave, Master => "Modbus_Send_Receive".Extrusora_3.Master, SP_Out => "Modbus_Send_Receive".Extrusora_3.SP, PV_Out => "Modbus_Send_Receive".Extrusora_3.PV, Malfunction => "Modbus_Send_Receive".Malfunction_3)
   END_RUNG
   // the same network as SCL:
   "Word_2_Bool"("1_registrador_in" := "Modbus_Send_Receive_1".Reading_Struct."32013",
                 "2_registrador_in" := "Modbus_Send_Receive_1".Reading_Struct."32014",
                 "3_registrador_in" := "Modbus_Send_Receive_1".Reading_Struct."32015",
                 "4_registrador_in" := "Modbus_Send_Receive_1".Reading_Struct."32016",
                 "5_registrador_in" := "Modbus_Send_Receive_1".Reading_Struct."32017",
                 Fancoil_Ligado => "Modbus_Send_Receive".Extrusora_3.Ligado,
                 Heating => "Modbus_Send_Receive".Extrusora_3.Heating,
                 Cooling => "Modbus_Send_Receive".Extrusora_3.Cooling,
                 Fan => "Modbus_Send_Receive".Extrusora_3.Fan,
                 Sts_Fan => "Modbus_Send_Receive".Extrusora_3.Sts_Fan,
                 Sts_Heating => "Modbus_Send_Receive".Extrusora_3.Sts_Heating,
                 Sts_Cooling => "Modbus_Send_Receive".Extrusora_3.Sts_Cooling,
                 Slave => "Modbus_Send_Receive".Extrusora_3.Slave,
                 Master => "Modbus_Send_Receive".Extrusora_3.Master,
                 SP_Out => "Modbus_Send_Receive".Extrusora_3.SP,
                 PV_Out => "Modbus_Send_Receive".Extrusora_3.PV,
                 Malfunction => "Modbus_Send_Receive".Malfunction_3);
END_REGION

REGION Network 4: Extrusora 4
   RUNG wire#powerrail
      "Word_2_Bool"("1_registrador_in" := "Modbus_Send_Receive_1".Reading_Struct."32019", "2_registrador_in" := "Modbus_Send_Receive_1".Reading_Struct."32020", "3_registrador_in" := "Modbus_Send_Receive_1".Reading_Struct."32021", "4_registrador_in" := "Modbus_Send_Receive_1".Reading_Struct."32022", "5_registrador_in" := "Modbus_Send_Receive_1".Reading_Struct."32023", Fancoil_Ligado => "Modbus_Send_Receive".Extrusora_4.Ligado, Heating => "Modbus_Send_Receive".Extrusora_4.Heating, Cooling => "Modbus_Send_Receive".Extrusora_4.Cooling, Fan => "Modbus_Send_Receive".Extrusora_4.Fan, Sts_Fan => "Modbus_Send_Receive".Extrusora_4.Sts_Fan, Sts_Heating => "Modbus_Send_Receive".Extrusora_4.Sts_Heating, Sts_Cooling => "Modbus_Send_Receive".Extrusora_4.Sts_Cooling, Slave => "Modbus_Send_Receive".Extrusora_4.Slave, Master => "Modbus_Send_Receive".Extrusora_4.Master, SP_Out => "Modbus_Send_Receive".Extrusora_4.SP, PV_Out => "Modbus_Send_Receive".Extrusora_4.PV, Malfunction => "Modbus_Send_Receive".Malfunction_4)
   END_RUNG
   // the same network as SCL:
   "Word_2_Bool"("1_registrador_in" := "Modbus_Send_Receive_1".Reading_Struct."32019",
                 "2_registrador_in" := "Modbus_Send_Receive_1".Reading_Struct."32020",
                 "3_registrador_in" := "Modbus_Send_Receive_1".Reading_Struct."32021",
                 "4_registrador_in" := "Modbus_Send_Receive_1".Reading_Struct."32022",
                 "5_registrador_in" := "Modbus_Send_Receive_1".Reading_Struct."32023",
                 Fancoil_Ligado => "Modbus_Send_Receive".Extrusora_4.Ligado,
                 Heating => "Modbus_Send_Receive".Extrusora_4.Heating,
                 Cooling => "Modbus_Send_Receive".Extrusora_4.Cooling,
                 Fan => "Modbus_Send_Receive".Extrusora_4.Fan,
                 Sts_Fan => "Modbus_Send_Receive".Extrusora_4.Sts_Fan,
                 Sts_Heating => "Modbus_Send_Receive".Extrusora_4.Sts_Heating,
                 Sts_Cooling => "Modbus_Send_Receive".Extrusora_4.Sts_Cooling,
                 Slave => "Modbus_Send_Receive".Extrusora_4.Slave,
                 Master => "Modbus_Send_Receive".Extrusora_4.Master,
                 SP_Out => "Modbus_Send_Receive".Extrusora_4.SP,
                 PV_Out => "Modbus_Send_Receive".Extrusora_4.PV,
                 Malfunction => "Modbus_Send_Receive".Malfunction_4);
END_REGION

REGION Network 5: Extrusora 5
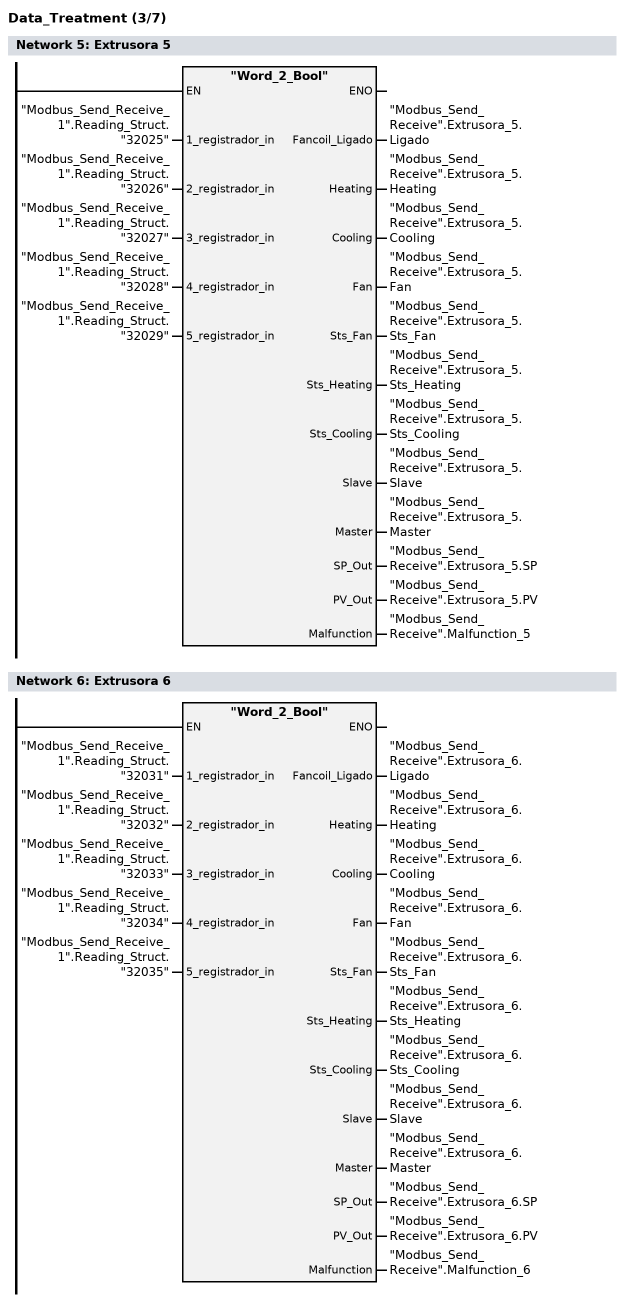
   RUNG wire#powerrail
      "Word_2_Bool"("1_registrador_in" := "Modbus_Send_Receive_1".Reading_Struct."32025", "2_registrador_in" := "Modbus_Send_Receive_1".Reading_Struct."32026", "3_registrador_in" := "Modbus_Send_Receive_1".Reading_Struct."32027", "4_registrador_in" := "Modbus_Send_Receive_1".Reading_Struct."32028", "5_registrador_in" := "Modbus_Send_Receive_1".Reading_Struct."32029", Fancoil_Ligado => "Modbus_Send_Receive".Extrusora_5.Ligado, Heating => "Modbus_Send_Receive".Extrusora_5.Heating, Cooling => "Modbus_Send_Receive".Extrusora_5.Cooling, Fan => "Modbus_Send_Receive".Extrusora_5.Fan, Sts_Fan => "Modbus_Send_Receive".Extrusora_5.Sts_Fan, Sts_Heating => "Modbus_Send_Receive".Extrusora_5.Sts_Heating, Sts_Cooling => "Modbus_Send_Receive".Extrusora_5.Sts_Cooling, Slave => "Modbus_Send_Receive".Extrusora_5.Slave, Master => "Modbus_Send_Receive".Extrusora_5.Master, SP_Out => "Modbus_Send_Receive".Extrusora_5.SP, PV_Out => "Modbus_Send_Receive".Extrusora_5.PV, Malfunction => "Modbus_Send_Receive".Malfunction_5)
   END_RUNG
   // the same network as SCL:
   "Word_2_Bool"("1_registrador_in" := "Modbus_Send_Receive_1".Reading_Struct."32025",
                 "2_registrador_in" := "Modbus_Send_Receive_1".Reading_Struct."32026",
                 "3_registrador_in" := "Modbus_Send_Receive_1".Reading_Struct."32027",
                 "4_registrador_in" := "Modbus_Send_Receive_1".Reading_Struct."32028",
                 "5_registrador_in" := "Modbus_Send_Receive_1".Reading_Struct."32029",
                 Fancoil_Ligado => "Modbus_Send_Receive".Extrusora_5.Ligado,
                 Heating => "Modbus_Send_Receive".Extrusora_5.Heating,
                 Cooling => "Modbus_Send_Receive".Extrusora_5.Cooling,
                 Fan => "Modbus_Send_Receive".Extrusora_5.Fan,
                 Sts_Fan => "Modbus_Send_Receive".Extrusora_5.Sts_Fan,
                 Sts_Heating => "Modbus_Send_Receive".Extrusora_5.Sts_Heating,
                 Sts_Cooling => "Modbus_Send_Receive".Extrusora_5.Sts_Cooling,
                 Slave => "Modbus_Send_Receive".Extrusora_5.Slave,
                 Master => "Modbus_Send_Receive".Extrusora_5.Master,
                 SP_Out => "Modbus_Send_Receive".Extrusora_5.SP,
                 PV_Out => "Modbus_Send_Receive".Extrusora_5.PV,
                 Malfunction => "Modbus_Send_Receive".Malfunction_5);
END_REGION

REGION Network 6: Extrusora 6
   RUNG wire#powerrail
      "Word_2_Bool"("1_registrador_in" := "Modbus_Send_Receive_1".Reading_Struct."32031", "2_registrador_in" := "Modbus_Send_Receive_1".Reading_Struct."32032", "3_registrador_in" := "Modbus_Send_Receive_1".Reading_Struct."32033", "4_registrador_in" := "Modbus_Send_Receive_1".Reading_Struct."32034", "5_registrador_in" := "Modbus_Send_Receive_1".Reading_Struct."32035", Fancoil_Ligado => "Modbus_Send_Receive".Extrusora_6.Ligado, Heating => "Modbus_Send_Receive".Extrusora_6.Heating, Cooling => "Modbus_Send_Receive".Extrusora_6.Cooling, Fan => "Modbus_Send_Receive".Extrusora_6.Fan, Sts_Fan => "Modbus_Send_Receive".Extrusora_6.Sts_Fan, Sts_Heating => "Modbus_Send_Receive".Extrusora_6.Sts_Heating, Sts_Cooling => "Modbus_Send_Receive".Extrusora_6.Sts_Cooling, Slave => "Modbus_Send_Receive".Extrusora_6.Slave, Master => "Modbus_Send_Receive".Extrusora_6.Master, SP_Out => "Modbus_Send_Receive".Extrusora_6.SP, PV_Out => "Modbus_Send_Receive".Extrusora_6.PV, Malfunction => "Modbus_Send_Receive".Malfunction_6)
   END_RUNG
   // the same network as SCL:
   "Word_2_Bool"("1_registrador_in" := "Modbus_Send_Receive_1".Reading_Struct."32031",
                 "2_registrador_in" := "Modbus_Send_Receive_1".Reading_Struct."32032",
                 "3_registrador_in" := "Modbus_Send_Receive_1".Reading_Struct."32033",
                 "4_registrador_in" := "Modbus_Send_Receive_1".Reading_Struct."32034",
                 "5_registrador_in" := "Modbus_Send_Receive_1".Reading_Struct."32035",
                 Fancoil_Ligado => "Modbus_Send_Receive".Extrusora_6.Ligado,
                 Heating => "Modbus_Send_Receive".Extrusora_6.Heating,
                 Cooling => "Modbus_Send_Receive".Extrusora_6.Cooling,
                 Fan => "Modbus_Send_Receive".Extrusora_6.Fan,
                 Sts_Fan => "Modbus_Send_Receive".Extrusora_6.Sts_Fan,
                 Sts_Heating => "Modbus_Send_Receive".Extrusora_6.Sts_Heating,
                 Sts_Cooling => "Modbus_Send_Receive".Extrusora_6.Sts_Cooling,
                 Slave => "Modbus_Send_Receive".Extrusora_6.Slave,
                 Master => "Modbus_Send_Receive".Extrusora_6.Master,
                 SP_Out => "Modbus_Send_Receive".Extrusora_6.SP,
                 PV_Out => "Modbus_Send_Receive".Extrusora_6.PV,
                 Malfunction => "Modbus_Send_Receive".Malfunction_6);
END_REGION

REGION Network 7: Extrusora 8
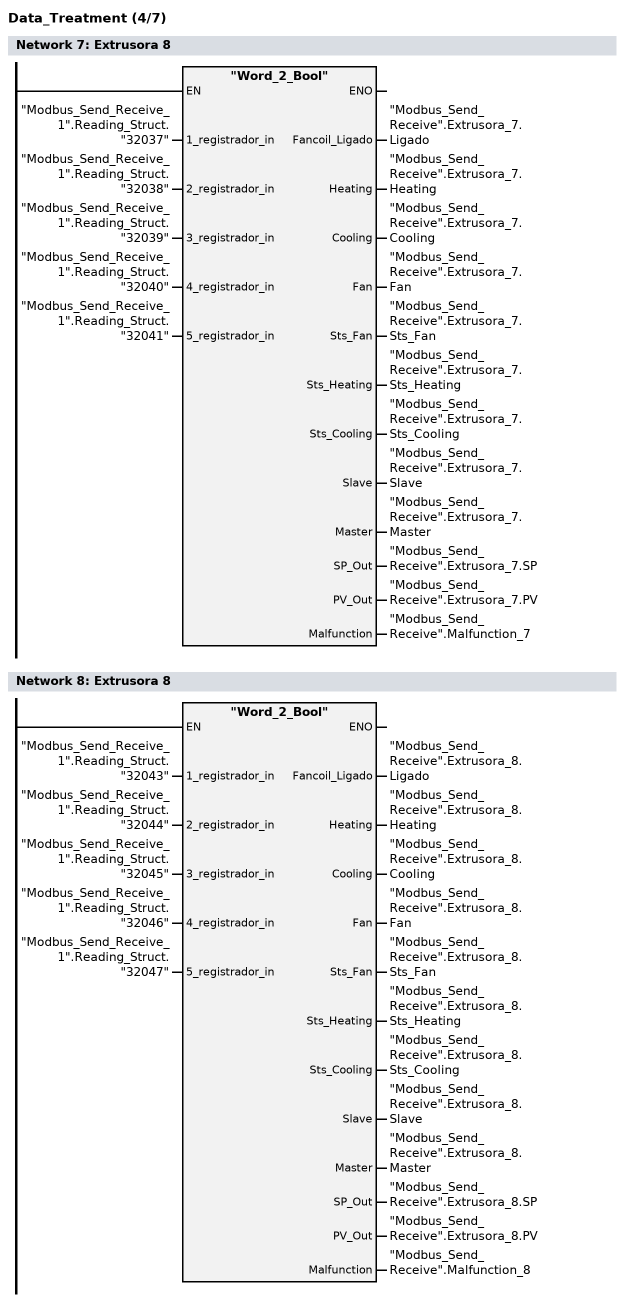
   RUNG wire#powerrail
      "Word_2_Bool"("1_registrador_in" := "Modbus_Send_Receive_1".Reading_Struct."32037", "2_registrador_in" := "Modbus_Send_Receive_1".Reading_Struct."32038", "3_registrador_in" := "Modbus_Send_Receive_1".Reading_Struct."32039", "4_registrador_in" := "Modbus_Send_Receive_1".Reading_Struct."32040", "5_registrador_in" := "Modbus_Send_Receive_1".Reading_Struct."32041", Fancoil_Ligado => "Modbus_Send_Receive".Extrusora_7.Ligado, Heating => "Modbus_Send_Receive".Extrusora_7.Heating, Cooling => "Modbus_Send_Receive".Extrusora_7.Cooling, Fan => "Modbus_Send_Receive".Extrusora_7.Fan, Sts_Fan => "Modbus_Send_Receive".Extrusora_7.Sts_Fan, Sts_Heating => "Modbus_Send_Receive".Extrusora_7.Sts_Heating, Sts_Cooling => "Modbus_Send_Receive".Extrusora_7.Sts_Cooling, Slave => "Modbus_Send_Receive".Extrusora_7.Slave, Master => "Modbus_Send_Receive".Extrusora_7.Master, SP_Out => "Modbus_Send_Receive".Extrusora_7.SP, PV_Out => "Modbus_Send_Receive".Extrusora_7.PV, Malfunction => "Modbus_Send_Receive".Malfunction_7)
   END_RUNG
   // the same network as SCL:
   "Word_2_Bool"("1_registrador_in" := "Modbus_Send_Receive_1".Reading_Struct."32037",
                 "2_registrador_in" := "Modbus_Send_Receive_1".Reading_Struct."32038",
                 "3_registrador_in" := "Modbus_Send_Receive_1".Reading_Struct."32039",
                 "4_registrador_in" := "Modbus_Send_Receive_1".Reading_Struct."32040",
                 "5_registrador_in" := "Modbus_Send_Receive_1".Reading_Struct."32041",
                 Fancoil_Ligado => "Modbus_Send_Receive".Extrusora_7.Ligado,
                 Heating => "Modbus_Send_Receive".Extrusora_7.Heating,
                 Cooling => "Modbus_Send_Receive".Extrusora_7.Cooling,
                 Fan => "Modbus_Send_Receive".Extrusora_7.Fan,
                 Sts_Fan => "Modbus_Send_Receive".Extrusora_7.Sts_Fan,
                 Sts_Heating => "Modbus_Send_Receive".Extrusora_7.Sts_Heating,
                 Sts_Cooling => "Modbus_Send_Receive".Extrusora_7.Sts_Cooling,
                 Slave => "Modbus_Send_Receive".Extrusora_7.Slave,
                 Master => "Modbus_Send_Receive".Extrusora_7.Master,
                 SP_Out => "Modbus_Send_Receive".Extrusora_7.SP,
                 PV_Out => "Modbus_Send_Receive".Extrusora_7.PV,
                 Malfunction => "Modbus_Send_Receive".Malfunction_7);
END_REGION

REGION Network 8: Extrusora 8
   RUNG wire#powerrail
      "Word_2_Bool"("1_registrador_in" := "Modbus_Send_Receive_1".Reading_Struct."32043", "2_registrador_in" := "Modbus_Send_Receive_1".Reading_Struct."32044", "3_registrador_in" := "Modbus_Send_Receive_1".Reading_Struct."32045", "4_registrador_in" := "Modbus_Send_Receive_1".Reading_Struct."32046", "5_registrador_in" := "Modbus_Send_Receive_1".Reading_Struct."32047", Fancoil_Ligado => "Modbus_Send_Receive".Extrusora_8.Ligado, Heating => "Modbus_Send_Receive".Extrusora_8.Heating, Cooling => "Modbus_Send_Receive".Extrusora_8.Cooling, Fan => "Modbus_Send_Receive".Extrusora_8.Fan, Sts_Fan => "Modbus_Send_Receive".Extrusora_8.Sts_Fan, Sts_Heating => "Modbus_Send_Receive".Extrusora_8.Sts_Heating, Sts_Cooling => "Modbus_Send_Receive".Extrusora_8.Sts_Cooling, Slave => "Modbus_Send_Receive".Extrusora_8.Slave, Master => "Modbus_Send_Receive".Extrusora_8.Master, SP_Out => "Modbus_Send_Receive".Extrusora_8.SP, PV_Out => "Modbus_Send_Receive".Extrusora_8.PV, Malfunction => "Modbus_Send_Receive".Malfunction_8)
   END_RUNG
   // the same network as SCL:
   "Word_2_Bool"("1_registrador_in" := "Modbus_Send_Receive_1".Reading_Struct."32043",
                 "2_registrador_in" := "Modbus_Send_Receive_1".Reading_Struct."32044",
                 "3_registrador_in" := "Modbus_Send_Receive_1".Reading_Struct."32045",
                 "4_registrador_in" := "Modbus_Send_Receive_1".Reading_Struct."32046",
                 "5_registrador_in" := "Modbus_Send_Receive_1".Reading_Struct."32047",
                 Fancoil_Ligado => "Modbus_Send_Receive".Extrusora_8.Ligado,
                 Heating => "Modbus_Send_Receive".Extrusora_8.Heating,
                 Cooling => "Modbus_Send_Receive".Extrusora_8.Cooling,
                 Fan => "Modbus_Send_Receive".Extrusora_8.Fan,
                 Sts_Fan => "Modbus_Send_Receive".Extrusora_8.Sts_Fan,
                 Sts_Heating => "Modbus_Send_Receive".Extrusora_8.Sts_Heating,
                 Sts_Cooling => "Modbus_Send_Receive".Extrusora_8.Sts_Cooling,
                 Slave => "Modbus_Send_Receive".Extrusora_8.Slave,
                 Master => "Modbus_Send_Receive".Extrusora_8.Master,
                 SP_Out => "Modbus_Send_Receive".Extrusora_8.SP,
                 PV_Out => "Modbus_Send_Receive".Extrusora_8.PV,
                 Malfunction => "Modbus_Send_Receive".Malfunction_8);
END_REGION

REGION Network 9: Extrusora 9
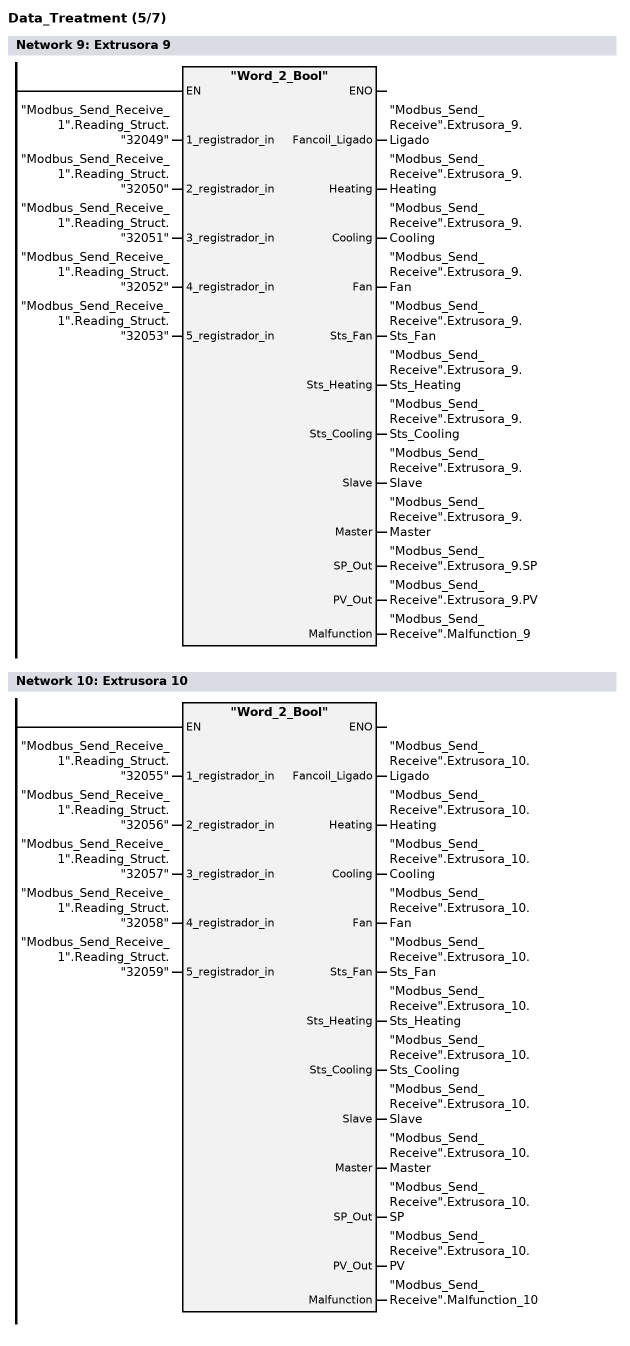
   RUNG wire#powerrail
      "Word_2_Bool"("1_registrador_in" := "Modbus_Send_Receive_1".Reading_Struct."32049", "2_registrador_in" := "Modbus_Send_Receive_1".Reading_Struct."32050", "3_registrador_in" := "Modbus_Send_Receive_1".Reading_Struct."32051", "4_registrador_in" := "Modbus_Send_Receive_1".Reading_Struct."32052", "5_registrador_in" := "Modbus_Send_Receive_1".Reading_Struct."32053", Fancoil_Ligado => "Modbus_Send_Receive".Extrusora_9.Ligado, Heating => "Modbus_Send_Receive".Extrusora_9.Heating, Cooling => "Modbus_Send_Receive".Extrusora_9.Cooling, Fan => "Modbus_Send_Receive".Extrusora_9.Fan, Sts_Fan => "Modbus_Send_Receive".Extrusora_9.Sts_Fan, Sts_Heating => "Modbus_Send_Receive".Extrusora_9.Sts_Heating, Sts_Cooling => "Modbus_Send_Receive".Extrusora_9.Sts_Cooling, Slave => "Modbus_Send_Receive".Extrusora_9.Slave, Master => "Modbus_Send_Receive".Extrusora_9.Master, SP_Out => "Modbus_Send_Receive".Extrusora_9.SP, PV_Out => "Modbus_Send_Receive".Extrusora_9.PV, Malfunction => "Modbus_Send_Receive".Malfunction_9)
   END_RUNG
   // the same network as SCL:
   "Word_2_Bool"("1_registrador_in" := "Modbus_Send_Receive_1".Reading_Struct."32049",
                 "2_registrador_in" := "Modbus_Send_Receive_1".Reading_Struct."32050",
                 "3_registrador_in" := "Modbus_Send_Receive_1".Reading_Struct."32051",
                 "4_registrador_in" := "Modbus_Send_Receive_1".Reading_Struct."32052",
                 "5_registrador_in" := "Modbus_Send_Receive_1".Reading_Struct."32053",
                 Fancoil_Ligado => "Modbus_Send_Receive".Extrusora_9.Ligado,
                 Heating => "Modbus_Send_Receive".Extrusora_9.Heating,
                 Cooling => "Modbus_Send_Receive".Extrusora_9.Cooling,
                 Fan => "Modbus_Send_Receive".Extrusora_9.Fan,
                 Sts_Fan => "Modbus_Send_Receive".Extrusora_9.Sts_Fan,
                 Sts_Heating => "Modbus_Send_Receive".Extrusora_9.Sts_Heating,
                 Sts_Cooling => "Modbus_Send_Receive".Extrusora_9.Sts_Cooling,
                 Slave => "Modbus_Send_Receive".Extrusora_9.Slave,
                 Master => "Modbus_Send_Receive".Extrusora_9.Master,
                 SP_Out => "Modbus_Send_Receive".Extrusora_9.SP,
                 PV_Out => "Modbus_Send_Receive".Extrusora_9.PV,
                 Malfunction => "Modbus_Send_Receive".Malfunction_9);
END_REGION

REGION Network 10: Extrusora 10
   RUNG wire#powerrail
      "Word_2_Bool"("1_registrador_in" := "Modbus_Send_Receive_1".Reading_Struct."32055", "2_registrador_in" := "Modbus_Send_Receive_1".Reading_Struct."32056", "3_registrador_in" := "Modbus_Send_Receive_1".Reading_Struct."32057", "4_registrador_in" := "Modbus_Send_Receive_1".Reading_Struct."32058", "5_registrador_in" := "Modbus_Send_Receive_1".Reading_Struct."32059", Fancoil_Ligado => "Modbus_Send_Receive".Extrusora_10.Ligado, Heating => "Modbus_Send_Receive".Extrusora_10.Heating, Cooling => "Modbus_Send_Receive".Extrusora_10.Cooling, Fan => "Modbus_Send_Receive".Extrusora_10.Fan, Sts_Fan => "Modbus_Send_Receive".Extrusora_10.Sts_Fan, Sts_Heating => "Modbus_Send_Receive".Extrusora_10.Sts_Heating, Sts_Cooling => "Modbus_Send_Receive".Extrusora_10.Sts_Cooling, Slave => "Modbus_Send_Receive".Extrusora_10.Slave, Master => "Modbus_Send_Receive".Extrusora_10.Master, SP_Out => "Modbus_Send_Receive".Extrusora_10.SP, PV_Out => "Modbus_Send_Receive".Extrusora_10.PV, Malfunction => "Modbus_Send_Receive".Malfunction_10)
   END_RUNG
   // the same network as SCL:
   "Word_2_Bool"("1_registrador_in" := "Modbus_Send_Receive_1".Reading_Struct."32055",
                 "2_registrador_in" := "Modbus_Send_Receive_1".Reading_Struct."32056",
                 "3_registrador_in" := "Modbus_Send_Receive_1".Reading_Struct."32057",
                 "4_registrador_in" := "Modbus_Send_Receive_1".Reading_Struct."32058",
                 "5_registrador_in" := "Modbus_Send_Receive_1".Reading_Struct."32059",
                 Fancoil_Ligado => "Modbus_Send_Receive".Extrusora_10.Ligado,
                 Heating => "Modbus_Send_Receive".Extrusora_10.Heating,
                 Cooling => "Modbus_Send_Receive".Extrusora_10.Cooling,
                 Fan => "Modbus_Send_Receive".Extrusora_10.Fan,
                 Sts_Fan => "Modbus_Send_Receive".Extrusora_10.Sts_Fan,
                 Sts_Heating => "Modbus_Send_Receive".Extrusora_10.Sts_Heating,
                 Sts_Cooling => "Modbus_Send_Receive".Extrusora_10.Sts_Cooling,
                 Slave => "Modbus_Send_Receive".Extrusora_10.Slave,
                 Master => "Modbus_Send_Receive".Extrusora_10.Master,
                 SP_Out => "Modbus_Send_Receive".Extrusora_10.SP,
                 PV_Out => "Modbus_Send_Receive".Extrusora_10.PV,
                 Malfunction => "Modbus_Send_Receive".Malfunction_10);
END_REGION

